Module[2].Input.SkillInput[14].ParameterInput[2] := Module2002.Input.SkillInput.SkillInput14.ParameterInput.ParameterInput2;
Module2002.Output.SkillOutput.SkillOutput14.ParameterOutput.ParameterOutput2 := Module[2].Output.SkillOutput[14].ParameterOutput[2];
Module[2].Input.SkillInput[14].ParameterInput[3] := Module2002.Input.SkillInput.SkillInput14.ParameterInput.ParameterInput3;
Module2002.Output.SkillOutput.SkillOutput14.ParameterOutput.ParameterOutput3 := Module[2].Output.SkillOutput[14].ParameterOutput[3];
Module[2].Input.SkillInput[14].ParameterInput[4] := Module2002.Input.SkillInput.SkillInput14.ParameterInput.ParameterInput4;
Module2002.Output.SkillOutput.SkillOutput14.ParameterOutput.ParameterOutput4 := Module[2].Output.SkillOutput[14].ParameterOutput[4];
Module[2].Input.SkillInput[14].ParameterInput[5] := Module2002.Input.SkillInput.SkillInput14.ParameterInput.ParameterInput5;
Module2002.Output.SkillOutput.SkillOutput14.ParameterOutput.ParameterOutput5 := Module[2].Output.SkillOutput[14].ParameterOutput[5];
Module[2].Input.SkillInput[15].Execute := Module2002.Input.SkillInput.SkillInput15.Execute;
Module2002.Output.SkillOutput.SkillOutput15.Dummy := Module[2].Output.SkillOutput[15].Dummy;
Module2002.Output.SkillOutput.SkillOutput15.ID := Module[2].Output.SkillOutput[15].ID;
Module2002.Output.SkillOutput.SkillOutput15.Name := Module[2].Output.SkillOutput[15].Name;
Module2002.Output.SkillOutput.SkillOutput15.Activated := Module[2].Output.SkillOutput[15].Activated;
Module2002.Output.SkillOutput.SkillOutput15.Ready := Module[2].Output.SkillOutput[15].Ready;
Module2002.Output.SkillOutput.SkillOutput15.Busy := Module[2].Output.SkillOutput[15].Busy;
Module2002.Output.SkillOutput.SkillOutput15.Done := Module[2].Output.SkillOutput[15].Done;
Module2002.Output.SkillOutput.SkillOutput15.Error := Module[2].Output.SkillOutput[15].Error;
Module2002.Output.Statevalue.Statevalue0 := Module[2].Output.Statevalue[0];
Module2002.Output.Statevalue.Statevalue1 := Module[2].Output.Statevalue[1];
Module2002.Output.Statevalue.Statevalue2 := Module[2].Output.Statevalue[2];
Module2002.Output.Statevalue.Statevalue3 := Module[2].Output.Statevalue[3];
Module2002.Output.Statevalue.Statevalue4 := Module[2].Output.Statevalue[4];
Module2002.Output.Statevalue.Statevalue5 := Module[2].Output.Statevalue[5];
Module2002.Output.Statevalue.Statevalue6 := Module[2].Output.Statevalue[6];
Module2002.Output.Statevalue.Statevalue7 := Module[2].Output.Statevalue[7];
Module2002.Output.Statevalue.Statevalue8 := Module[2].Output.Statevalue[8];
Module2002.Output.Statevalue.Statevalue9 := Module[2].Output.Statevalue[9];
Module2002.Output.Statevalue.Statevalue10 := Module[2].Output.Statevalue[10];
Module[2].Input.SkillInput[15].ParameterInput[0] := Module2002.Input.SkillInput.SkillInput15.ParameterInput.ParameterInput0;
Module2002.Output.SkillOutput.SkillOutput15.ParameterOutput.ParameterOutput0 := Module[2].Output.SkillOutput[15].ParameterOutput[0];
Module[2].Input.SkillInput[15].ParameterInput[1] := Module2002.Input.SkillInput.SkillInput15.ParameterInput.ParameterInput1;
Module2002.Output.SkillOutput.SkillOutput15.ParameterOutput.ParameterOutput1 := Module[2].Output.SkillOutput[15].ParameterOutput[1];
Module[2].Input.SkillInput[15].ParameterInput[2] := Module2002.Input.SkillInput.SkillInput15.ParameterInput.ParameterInput2;
Module2002.Output.SkillOutput.SkillOutput15.ParameterOutput.ParameterOutput2 := Module[2].Output.SkillOutput[15].ParameterOutput[2];
Module[2].Input.SkillInput[15].ParameterInput[3] := Module2002.Input.SkillInput.SkillInput15.ParameterInput.ParameterInput3;
Module2002.Output.SkillOutput.SkillOutput15.ParameterOutput.ParameterOutput3 := Module[2].Output.SkillOutput[15].ParameterOutput[3];
Module[2].Input.SkillInput[15].ParameterInput[4] := Module2002.Input.SkillInput.SkillInput15.ParameterInput.ParameterInput4;
Module2002.Output.SkillOutput.SkillOutput15.ParameterOutput.ParameterOutput4 := Module[2].Output.SkillOutput[15].ParameterOutput[4];
Module[2].Input.SkillInput[15].ParameterInput[5] := Module2002.Input.SkillInput.SkillInput15.ParameterInput.ParameterInput5;
Module2002.Output.SkillOutput.SkillOutput15.ParameterOutput.ParameterOutput5 := Module[2].Output.SkillOutput[15].ParameterOutput[5];
Module[3].Input.Mode := Module2003.Input.Mode;
Module[3].Input.ConnectionTestInput := Module2003.Input.ConnectionTestInput;
Module[3].Input.PositionInput := Module2003.Input.PositionInput;
Module[3].Input.Watchbit := Module2003.Input.Watchbit;
Module[3].Input.EmergencyStop := Module2003.Input.EmergencyStop;
Module2003.Output.Dummy := Module[3].Output.Dummy;
Module2003.Output.Name := Module[3].Output.Name;
Module2003.Output.ID := Module[3].Output.ID;
Module2003.Output.IP := Module[3].Output.IP;
Module2003.Output.Idle := Module[3].Output.Idle;
Module2003.Output.Connected := Module[3].Output.Connected;
Module2003.Output.Error := Module[3].Output.Error;
Module2003.Output.ErrorID := Module[3].Output.ErrorID;
Module2003.Output.ErrorDescription := Module[3].Output.ErrorDescription;
Module2003.Output.CurrentTaskDescription := Module[3].Output.CurrentTaskDescription;
Module2003.Output.PositionSensor := Module[3].Output.PositionSensor;
Module2003.Output.ConnectionTestOutput := Module[3].Output.ConnectionTestOutput;
Module[3].Input.SkillInput[0].Execute := Module2003.Input.SkillInput.SkillInput0.Execute;
Module2003.Output.SkillOutput.SkillOutput0.Dummy := Module[3].Output.SkillOutput[0].Dummy;
Module2003.Output.SkillOutput.SkillOutput0.ID := Module[3].Output.SkillOutput[0].ID;
Module2003.Output.SkillOutput.SkillOutput0.Name := Module[3].Output.SkillOutput[0].Name;
Module2003.Output.SkillOutput.SkillOutput0.Activated := Module[3].Output.SkillOutput[0].Activated;
Module2003.Output.SkillOutput.SkillOutput0.Ready := Module[3].Output.SkillOutput[0].Ready;
Module2003.Output.SkillOutput.SkillOutput0.Busy := Module[3].Output.SkillOutput[0].Busy;
Module2003.Output.SkillOutput.SkillOutput0.Done := Module[3].Output.SkillOutput[0].Done;
Module2003.Output.SkillOutput.SkillOutput0.Error := Module[3].Output.SkillOutput[0].Error;
Module2003.Output.Statevalue.Statevalue0 := Module[3].Output.Statevalue[0];
Module2003.Output.Statevalue.Statevalue1 := Module[3].Output.Statevalue[1];
Module2003.Output.Statevalue.Statevalue2 := Module[3].Output.Statevalue[2];
Module2003.Output.Statevalue.Statevalue3 := Module[3].Output.Statevalue[3];
Module2003.Output.Statevalue.Statevalue4 := Module[3].Output.Statevalue[4];
Module2003.Output.Statevalue.Statevalue5 := Module[3].Output.Statevalue[5];
Module2003.Output.Statevalue.Statevalue6 := Module[3].Output.Statevalue[6];
Module2003.Output.Statevalue.Statevalue7 := Module[3].Output.Statevalue[7];
Module2003.Output.Statevalue.Statevalue8 := Module[3].Output.Statevalue[8];
Module2003.Output.Statevalue.Statevalue9 := Module[3].Output.Statevalue[9];
Module2003.Output.Statevalue.Statevalue10 := Module[3].Output.Statevalue[10];
Module[3].Input.SkillInput[0].ParameterInput[0] := Module2003.Input.SkillInput.SkillInput0.ParameterInput.ParameterInput0;
Module2003.Output.SkillOutput.SkillOutput0.ParameterOutput.ParameterOutput0 := Module[3].Output.SkillOutput[0].ParameterOutput[0];
Module[3].Input.SkillInput[0].ParameterInput[1] := Module2003.Input.SkillInput.SkillInput0.ParameterInput.ParameterInput1;
Module2003.Output.SkillOutput.SkillOutput0.ParameterOutput.ParameterOutput1 := Module[3].Output.SkillOutput[0].ParameterOutput[1];
Module[3].Input.SkillInput[0].ParameterInput[2] := Module2003.Input.SkillInput.SkillInput0.ParameterInput.ParameterInput2;
Module2003.Output.SkillOutput.SkillOutput0.ParameterOutput.ParameterOutput2 := Module[3].Output.SkillOutput[0].ParameterOutput[2];
Module[3].Input.SkillInput[0].ParameterInput[3] := Module2003.Input.SkillInput.SkillInput0.ParameterInput.ParameterInput3;
Module2003.Output.SkillOutput.SkillOutput0.ParameterOutput.ParameterOutput3 := Module[3].Output.SkillOutput[0].ParameterOutput[3];
Module[3].Input.SkillInput[0].ParameterInput[4] := Module2003.Input.SkillInput.SkillInput0.ParameterInput.ParameterInput4;
Module2003.Output.SkillOutput.SkillOutput0.ParameterOutput.ParameterOutput4 := Module[3].Output.SkillOutput[0].ParameterOutput[4];
Module[3].Input.SkillInput[0].ParameterInput[5] := Module2003.Input.SkillInput.SkillInput0.ParameterInput.ParameterInput5;
Module2003.Output.SkillOutput.SkillOutput0.ParameterOutput.ParameterOutput5 := Module[3].Output.SkillOutput[0].ParameterOutput[5];
Module[3].Input.SkillInput[1].Execute := Module2003.Input.SkillInput.SkillInput1.Execute;
Module2003.Output.SkillOutput.SkillOutput1.Dummy := Module[3].Output.SkillOutput[1].Dummy;
Module2003.Output.SkillOutput.SkillOutput1.ID := Module[3].Output.SkillOutput[1].ID;
Module2003.Output.SkillOutput.SkillOutput1.Name := Module[3].Output.SkillOutput[1].Name;
Module2003.Output.SkillOutput.SkillOutput1.Activated := Module[3].Output.SkillOutput[1].Activated;
Module2003.Output.SkillOutput.SkillOutput1.Ready := Module[3].Output.SkillOutput[1].Ready;
Module2003.Output.SkillOutput.SkillOutput1.Busy := Module[3].Output.SkillOutput[1].Busy;
Module2003.Output.SkillOutput.SkillOutput1.Done := Module[3].Output.SkillOutput[1].Done;
Module2003.Output.SkillOutput.SkillOutput1.Error := Module[3].Output.SkillOutput[1].Error;
Module2003.Output.Statevalue.Statevalue0 := Module[3].Output.Statevalue[0];
Module2003.Output.Statevalue.Statevalue1 := Module[3].Output.Statevalue[1];
Module2003.Output.Statevalue.Statevalue2 := Module[3].Output.Statevalue[2];
Module2003.Output.Statevalue.Statevalue3 := Module[3].Output.Statevalue[3];
Module2003.Output.Statevalue.Statevalue4 := Module[3].Output.Statevalue[4];
Module2003.Output.Statevalue.Statevalue5 := Module[3].Output.Statevalue[5];
Module2003.Output.Statevalue.Statevalue6 := Module[3].Output.Statevalue[6];
Module2003.Output.Statevalue.Statevalue7 := Module[3].Output.Statevalue[7];
Module2003.Output.Statevalue.Statevalue8 := Module[3].Output.Statevalue[8];
Module2003.Output.Statevalue.Statevalue9 := Module[3].Output.Statevalue[9];
Module2003.Output.Statevalue.Statevalue10 := Module[3].Output.Statevalue[10];
Module[3].Input.SkillInput[1].ParameterInput[0] := Module2003.Input.SkillInput.SkillInput1.ParameterInput.ParameterInput0;
Module2003.Output.SkillOutput.SkillOutput1.ParameterOutput.ParameterOutput0 := Module[3].Output.SkillOutput[1].ParameterOutput[0];
Module[3].Input.SkillInput[1].ParameterInput[1] := Module2003.Input.SkillInput.SkillInput1.ParameterInput.ParameterInput1;
Module2003.Output.SkillOutput.SkillOutput1.ParameterOutput.ParameterOutput1 := Module[3].Output.SkillOutput[1].ParameterOutput[1];
Module[3].Input.SkillInput[1].ParameterInput[2] := Module2003.Input.SkillInput.SkillInput1.ParameterInput.ParameterInput2;
Module2003.Output.SkillOutput.SkillOutput1.ParameterOutput.ParameterOutput2 := Module[3].Output.SkillOutput[1].ParameterOutput[2];
Module[3].Input.SkillInput[1].ParameterInput[3] := Module2003.Input.SkillInput.SkillInput1.ParameterInput.ParameterInput3;
Module2003.Output.SkillOutput.SkillOutput1.ParameterOutput.ParameterOutput3 := Module[3].Output.SkillOutput[1].ParameterOutput[3];
Module[3].Input.SkillInput[1].ParameterInput[4] := Module2003.Input.SkillInput.SkillInput1.ParameterInput.ParameterInput4;
Module2003.Output.SkillOutput.SkillOutput1.ParameterOutput.ParameterOutput4 := Module[3].Output.SkillOutput[1].ParameterOutput[4];
Module[3].Input.SkillInput[1].ParameterInput[5] := Module2003.Input.SkillInput.SkillInput1.ParameterInput.ParameterInput5;
Module2003.Output.SkillOutput.SkillOutput1.ParameterOutput.ParameterOutput5 := Module[3].Output.SkillOutput[1].ParameterOutput[5];
Module[3].Input.SkillInput[2].Execute := Module2003.Input.SkillInput.SkillInput2.Execute;
Module2003.Output.SkillOutput.SkillOutput2.Dummy := Module[3].Output.SkillOutput[2].Dummy;
Module2003.Output.SkillOutput.SkillOutput2.ID := Module[3].Output.SkillOutput[2].ID;
Module2003.Output.SkillOutput.SkillOutput2.Name := Module[3].Output.SkillOutput[2].Name;
Module2003.Output.SkillOutput.SkillOutput2.Activated := Module[3].Output.SkillOutput[2].Activated;
Module2003.Output.SkillOutput.SkillOutput2.Ready := Module[3].Output.SkillOutput[2].Ready;
Module2003.Output.SkillOutput.SkillOutput2.Busy := Module[3].Output.SkillOutput[2].Busy;
Module2003.Output.SkillOutput.SkillOutput2.Done := Module[3].Output.SkillOutput[2].Done;
Module2003.Output.SkillOutput.SkillOutput2.Error := Module[3].Output.SkillOutput[2].Error;
Module2003.Output.Statevalue.Statevalue0 := Module[3].Output.Statevalue[0];
Module2003.Output.Statevalue.Statevalue1 := Module[3].Output.Statevalue[1];
Module2003.Output.Statevalue.Statevalue2 := Module[3].Output.Statevalue[2];
Module2003.Output.Statevalue.Statevalue3 := Module[3].Output.Statevalue[3];
Module2003.Output.Statevalue.Statevalue4 := Module[3].Output.Statevalue[4];
Module2003.Output.Statevalue.Statevalue5 := Module[3].Output.Statevalue[5];
Module2003.Output.Statevalue.Statevalue6 := Module[3].Output.Statevalue[6];
Module2003.Output.Statevalue.Statevalue7 := Module[3].Output.Statevalue[7];
Module2003.Output.Statevalue.Statevalue8 := Module[3].Output.Statevalue[8];
Module2003.Output.Statevalue.Statevalue9 := Module[3].Output.Statevalue[9];
Module2003.Output.Statevalue.Statevalue10 := Module[3].Output.Statevalue[10];
Module[3].Input.SkillInput[2].ParameterInput[0] := Module2003.Input.SkillInput.SkillInput2.ParameterInput.ParameterInput0;
Module2003.Output.SkillOutput.SkillOutput2.ParameterOutput.ParameterOutput0 := Module[3].Output.SkillOutput[2].ParameterOutput[0];
Module[3].Input.SkillInput[2].ParameterInput[1] := Module2003.Input.SkillInput.SkillInput2.ParameterInput.ParameterInput1;
Module2003.Output.SkillOutput.SkillOutput2.ParameterOutput.ParameterOutput1 := Module[3].Output.SkillOutput[2].ParameterOutput[1];
Module[3].Input.SkillInput[2].ParameterInput[2] := Module2003.Input.SkillInput.SkillInput2.ParameterInput.ParameterInput2;
Module2003.Output.SkillOutput.SkillOutput2.ParameterOutput.ParameterOutput2 := Module[3].Output.SkillOutput[2].ParameterOutput[2];
Module[3].Input.SkillInput[2].ParameterInput[3] := Module2003.Input.SkillInput.SkillInput2.ParameterInput.ParameterInput3;
Module2003.Output.SkillOutput.SkillOutput2.ParameterOutput.ParameterOutput3 := Module[3].Output.SkillOutput[2].ParameterOutput[3];
Module[3].Input.SkillInput[2].ParameterInput[4] := Module2003.Input.SkillInput.SkillInput2.ParameterInput.ParameterInput4;
Module2003.Output.SkillOutput.SkillOutput2.ParameterOutput.ParameterOutput4 := Module[3].Output.SkillOutput[2].ParameterOutput[4];
Module[3].Input.SkillInput[2].ParameterInput[5] := Module2003.Input.SkillInput.SkillInput2.ParameterInput.ParameterInput5;
Module2003.Output.SkillOutput.SkillOutput2.ParameterOutput.ParameterOutput5 := Module[3].Output.SkillOutput[2].ParameterOutput[5];
Module[3].Input.SkillInput[3].Execute := Module2003.Input.SkillInput.SkillInput3.Execute;
Module2003.Output.SkillOutput.SkillOutput3.Dummy := Module[3].Output.SkillOutput[3].Dummy;
Module2003.Output.SkillOutput.SkillOutput3.ID := Module[3].Output.SkillOutput[3].ID;
Module2003.Output.SkillOutput.SkillOutput3.Name := Module[3].Output.SkillOutput[3].Name;
Module2003.Output.SkillOutput.SkillOutput3.Activated := Module[3].Output.SkillOutput[3].Activated;
Module2003.Output.SkillOutput.SkillOutput3.Ready := Module[3].Output.SkillOutput[3].Ready;
Module2003.Output.SkillOutput.SkillOutput3.Busy := Module[3].Output.SkillOutput[3].Busy;
Module2003.Output.SkillOutput.SkillOutput3.Done := Module[3].Output.SkillOutput[3].Done;
Module2003.Output.SkillOutput.SkillOutput3.Error := Module[3].Output.SkillOutput[3].Error;
Module2003.Output.Statevalue.Statevalue0 := Module[3].Output.Statevalue[0];
Module2003.Output.Statevalue.Statevalue1 := Module[3].Output.Statevalue[1];
Module2003.Output.Statevalue.Statevalue2 := Module[3].Output.Statevalue[2];
Module2003.Output.Statevalue.Statevalue3 := Module[3].Output.Statevalue[3];
Module2003.Output.Statevalue.Statevalue4 := Module[3].Output.Statevalue[4];
Module2003.Output.Statevalue.Statevalue5 := Module[3].Output.Statevalue[5];
Module2003.Output.Statevalue.Statevalue6 := Module[3].Output.Statevalue[6];
Module2003.Output.Statevalue.Statevalue7 := Module[3].Output.Statevalue[7];
Module2003.Output.Statevalue.Statevalue8 := Module[3].Output.Statevalue[8];
Module2003.Output.Statevalue.Statevalue9 := Module[3].Output.Statevalue[9];
Module2003.Output.Statevalue.Statevalue10 := Module[3].Output.Statevalue[10];
Module[3].Input.SkillInput[3].ParameterInput[0] := Module2003.Input.SkillInput.SkillInput3.ParameterInput.ParameterInput0;
Module2003.Output.SkillOutput.SkillOutput3.ParameterOutput.ParameterOutput0 := Module[3].Output.SkillOutput[3].ParameterOutput[0];
Module[3].Input.SkillInput[3].ParameterInput[1] := Module2003.Input.SkillInput.SkillInput3.ParameterInput.ParameterInput1;
Module2003.Output.SkillOutput.SkillOutput3.ParameterOutput.ParameterOutput1 := Module[3].Output.SkillOutput[3].ParameterOutput[1];
Module[3].Input.SkillInput[3].ParameterInput[2] := Module2003.Input.SkillInput.SkillInput3.ParameterInput.ParameterInput2;
Module2003.Output.SkillOutput.SkillOutput3.ParameterOutput.ParameterOutput2 := Module[3].Output.SkillOutput[3].ParameterOutput[2];
Module[3].Input.SkillInput[3].ParameterInput[3] := Module2003.Input.SkillInput.SkillInput3.ParameterInput.ParameterInput3;
Module2003.Output.SkillOutput.SkillOutput3.ParameterOutput.ParameterOutput3 := Module[3].Output.SkillOutput[3].ParameterOutput[3];
Module[3].Input.SkillInput[3].ParameterInput[4] := Module2003.Input.SkillInput.SkillInput3.ParameterInput.ParameterInput4;
Module2003.Output.SkillOutput.SkillOutput3.ParameterOutput.ParameterOutput4 := Module[3].Output.SkillOutput[3].ParameterOutput[4];
Module[3].Input.SkillInput[3].ParameterInput[5] := Module2003.Input.SkillInput.SkillInput3.ParameterInput.ParameterInput5;
Module2003.Output.SkillOutput.SkillOutput3.ParameterOutput.ParameterOutput5 := Module[3].Output.SkillOutput[3].ParameterOutput[5];
Module[3].Input.SkillInput[4].Execute := Module2003.Input.SkillInput.SkillInput4.Execute;
Module2003.Output.SkillOutput.SkillOutput4.Dummy := Module[3].Output.SkillOutput[4].Dummy;
Module2003.Output.SkillOutput.SkillOutput4.ID := Module[3].Output.SkillOutput[4].ID;
Module2003.Output.SkillOutput.SkillOutput4.Name := Module[3].Output.SkillOutput[4].Name;
Module2003.Output.SkillOutput.SkillOutput4.Activated := Module[3].Output.SkillOutput[4].Activated;
Module2003.Output.SkillOutput.SkillOutput4.Ready := Module[3].Output.SkillOutput[4].Ready;
Module2003.Output.SkillOutput.SkillOutput4.Busy := Module[3].Output.SkillOutput[4].Busy;
Module2003.Output.SkillOutput.SkillOutput4.Done := Module[3].Output.SkillOutput[4].Done;
Module2003.Output.SkillOutput.SkillOutput4.Error := Module[3].Output.SkillOutput[4].Error;
Module2003.Output.Statevalue.Statevalue0 := Module[3].Output.Statevalue[0];
Module2003.Output.Statevalue.Statevalue1 := Module[3].Output.Statevalue[1];
Module2003.Output.Statevalue.Statevalue2 := Module[3].Output.Statevalue[2];
Module2003.Output.Statevalue.Statevalue3 := Module[3].Output.Statevalue[3];
Module2003.Output.Statevalue.Statevalue4 := Module[3].Output.Statevalue[4];
Module2003.Output.Statevalue.Statevalue5 := Module[3].Output.Statevalue[5];
Module2003.Output.Statevalue.Statevalue6 := Module[3].Output.Statevalue[6];
Module2003.Output.Statevalue.Statevalue7 := Module[3].Output.Statevalue[7];
Module2003.Output.Statevalue.Statevalue8 := Module[3].Output.Statevalue[8];
Module2003.Output.Statevalue.Statevalue9 := Module[3].Output.Statevalue[9];
Module2003.Output.Statevalue.Statevalue10 := Module[3].Output.Statevalue[10];
Module[3].Input.SkillInput[4].ParameterInput[0] := Module2003.Input.SkillInput.SkillInput4.ParameterInput.ParameterInput0;
Module2003.Output.SkillOutput.SkillOutput4.ParameterOutput.ParameterOutput0 := Module[3].Output.SkillOutput[4].ParameterOutput[0];
Module[3].Input.SkillInput[4].ParameterInput[1] := Module2003.Input.SkillInput.SkillInput4.ParameterInput.ParameterInput1;
Module2003.Output.SkillOutput.SkillOutput4.ParameterOutput.ParameterOutput1 := Module[3].Output.SkillOutput[4].ParameterOutput[1];
Module[3].Input.SkillInput[4].ParameterInput[2] := Module2003.Input.SkillInput.SkillInput4.ParameterInput.ParameterInput2;
Module2003.Output.SkillOutput.SkillOutput4.ParameterOutput.ParameterOutput2 := Module[3].Output.SkillOutput[4].ParameterOutput[2];
Module[3].Input.SkillInput[4].ParameterInput[3] := Module2003.Input.SkillInput.SkillInput4.ParameterInput.ParameterInput3;
Module2003.Output.SkillOutput.SkillOutput4.ParameterOutput.ParameterOutput3 := Module[3].Output.SkillOutput[4].ParameterOutput[3];
Module[3].Input.SkillInput[4].ParameterInput[4] := Module2003.Input.SkillInput.SkillInput4.ParameterInput.ParameterInput4;
Module2003.Output.SkillOutput.SkillOutput4.ParameterOutput.ParameterOutput4 := Module[3].Output.SkillOutput[4].ParameterOutput[4];
Module[3].Input.SkillInput[4].ParameterInput[5] := Module2003.Input.SkillInput.SkillInput4.ParameterInput.ParameterInput5;
Module2003.Output.SkillOutput.SkillOutput4.ParameterOutput.ParameterOutput5 := Module[3].Output.SkillOutput[4].ParameterOutput[5];
Module[3].Input.SkillInput[5].Execute := Module2003.Input.SkillInput.SkillInput5.Execute;
Module2003.Output.SkillOutput.SkillOutput5.Dummy := Module[3].Output.SkillOutput[5].Dummy;
Module2003.Output.SkillOutput.SkillOutput5.ID := Module[3].Output.SkillOutput[5].ID;
Module2003.Output.SkillOutput.SkillOutput5.Name := Module[3].Output.SkillOutput[5].Name;
Module2003.Output.SkillOutput.SkillOutput5.Activated := Module[3].Output.SkillOutput[5].Activated;
Module2003.Output.SkillOutput.SkillOutput5.Ready := Module[3].Output.SkillOutput[5].Ready;
Module2003.Output.SkillOutput.SkillOutput5.Busy := Module[3].Output.SkillOutput[5].Busy;
Module2003.Output.SkillOutput.SkillOutput5.Done := Module[3].Output.SkillOutput[5].Done;
Module2003.Output.SkillOutput.SkillOutput5.Error := Module[3].Output.SkillOutput[5].Error;
Module2003.Output.Statevalue.Statevalue0 := Module[3].Output.Statevalue[0];
Module2003.Output.Statevalue.Statevalue1 := Module[3].Output.Statevalue[1];
Module2003.Output.Statevalue.Statevalue2 := Module[3].Output.Statevalue[2];
Module2003.Output.Statevalue.Statevalue3 := Module[3].Output.Statevalue[3];
Module2003.Output.Statevalue.Statevalue4 := Module[3].Output.Statevalue[4];
Module2003.Output.Statevalue.Statevalue5 := Module[3].Output.Statevalue[5];
Module2003.Output.Statevalue.Statevalue6 := Module[3].Output.Statevalue[6];
Module2003.Output.Statevalue.Statevalue7 := Module[3].Output.Statevalue[7];
Module2003.Output.Statevalue.Statevalue8 := Module[3].Output.Statevalue[8];
Module2003.Output.Statevalue.Statevalue9 := Module[3].Output.Statevalue[9];
Module2003.Output.Statevalue.Statevalue10 := Module[3].Output.Statevalue[10];
Module[3].Input.SkillInput[5].ParameterInput[0] := Module2003.Input.SkillInput.SkillInput5.ParameterInput.ParameterInput0;
Module2003.Output.SkillOutput.SkillOutput5.ParameterOutput.ParameterOutput0 := Module[3].Output.SkillOutput[5].ParameterOutput[0];
Module[3].Input.SkillInput[5].ParameterInput[1] := Module2003.Input.SkillInput.SkillInput5.ParameterInput.ParameterInput1;
Module2003.Output.SkillOutput.SkillOutput5.ParameterOutput.ParameterOutput1 := Module[3].Output.SkillOutput[5].ParameterOutput[1];
Module[3].Input.SkillInput[5].ParameterInput[2] := Module2003.Input.SkillInput.SkillInput5.ParameterInput.ParameterInput2;
Module2003.Output.SkillOutput.SkillOutput5.ParameterOutput.ParameterOutput2 := Module[3].Output.SkillOutput[5].ParameterOutput[2];
Module[3].Input.SkillInput[5].ParameterInput[3] := Module2003.Input.SkillInput.SkillInput5.ParameterInput.ParameterInput3;
Module2003.Output.SkillOutput.SkillOutput5.ParameterOutput.ParameterOutput3 := Module[3].Output.SkillOutput[5].ParameterOutput[3];
Module[3].Input.SkillInput[5].ParameterInput[4] := Module2003.Input.SkillInput.SkillInput5.ParameterInput.ParameterInput4;
Module2003.Output.SkillOutput.SkillOutput5.ParameterOutput.ParameterOutput4 := Module[3].Output.SkillOutput[5].ParameterOutput[4];
Module[3].Input.SkillInput[5].ParameterInput[5] := Module2003.Input.SkillInput.SkillInput5.ParameterInput.ParameterInput5;
Module2003.Output.SkillOutput.SkillOutput5.ParameterOutput.ParameterOutput5 := Module[3].Output.SkillOutput[5].ParameterOutput[5];
Module[3].Input.SkillInput[6].Execute := Module2003.Input.SkillInput.SkillInput6.Execute;
Module2003.Output.SkillOutput.SkillOutput6.Dummy := Module[3].Output.SkillOutput[6].Dummy;
Module2003.Output.SkillOutput.SkillOutput6.ID := Module[3].Output.SkillOutput[6].ID;
Module2003.Output.SkillOutput.SkillOutput6.Name := Module[3].Output.SkillOutput[6].Name;
Module2003.Output.SkillOutput.SkillOutput6.Activated := Module[3].Output.SkillOutput[6].Activated;
Module2003.Output.SkillOutput.SkillOutput6.Ready := Module[3].Output.SkillOutput[6].Ready;
Module2003.Output.SkillOutput.SkillOutput6.Busy := Module[3].Output.SkillOutput[6].Busy;
Module2003.Output.SkillOutput.SkillOutput6.Done := Module[3].Output.SkillOutput[6].Done;
Module2003.Output.SkillOutput.SkillOutput6.Error := Module[3].Output.SkillOutput[6].Error;
Module2003.Output.Statevalue.Statevalue0 := Module[3].Output.Statevalue[0];
Module2003.Output.Statevalue.Statevalue1 := Module[3].Output.Statevalue[1];
Module2003.Output.Statevalue.Statevalue2 := Module[3].Output.Statevalue[2];
Module2003.Output.Statevalue.Statevalue3 := Module[3].Output.Statevalue[3];
Module2003.Output.Statevalue.Statevalue4 := Module[3].Output.Statevalue[4];
Module2003.Output.Statevalue.Statevalue5 := Module[3].Output.Statevalue[5];
Module2003.Output.Statevalue.Statevalue6 := Module[3].Output.Statevalue[6];
Module2003.Output.Statevalue.Statevalue7 := Module[3].Output.Statevalue[7];
Module2003.Output.Statevalue.Statevalue8 := Module[3].Output.Statevalue[8];
Module2003.Output.Statevalue.Statevalue9 := Module[3].Output.Statevalue[9];
Module2003.Output.Statevalue.Statevalue10 := Module[3].Output.Statevalue[10];
Module[3].Input.SkillInput[6].ParameterInput[0] := Module2003.Input.SkillInput.SkillInput6.ParameterInput.ParameterInput0;
Module2003.Output.SkillOutput.SkillOutput6.ParameterOutput.ParameterOutput0 := Module[3].Output.SkillOutput[6].ParameterOutput[0];
Module[3].Input.SkillInput[6].ParameterInput[1] := Module2003.Input.SkillInput.SkillInput6.ParameterInput.ParameterInput1;
Module2003.Output.SkillOutput.SkillOutput6.ParameterOutput.ParameterOutput1 := Module[3].Output.SkillOutput[6].ParameterOutput[1];
Module[3].Input.SkillInput[6].ParameterInput[2] := Module2003.Input.SkillInput.SkillInput6.ParameterInput.ParameterInput2;
Module2003.Output.SkillOutput.SkillOutput6.ParameterOutput.ParameterOutput2 := Module[3].Output.SkillOutput[6].ParameterOutput[2];
Module[3].Input.SkillInput[6].ParameterInput[3] := Module2003.Input.SkillInput.SkillInput6.ParameterInput.ParameterInput3;
Module2003.Output.SkillOutput.SkillOutput6.ParameterOutput.ParameterOutput3 := Module[3].Output.SkillOutput[6].ParameterOutput[3];
Module[3].Input.SkillInput[6].ParameterInput[4] := Module2003.Input.SkillInput.SkillInput6.ParameterInput.ParameterInput4;
Module2003.Output.SkillOutput.SkillOutput6.ParameterOutput.ParameterOutput4 := Module[3].Output.SkillOutput[6].ParameterOutput[4];
Module[3].Input.SkillInput[6].ParameterInput[5] := Module2003.Input.SkillInput.SkillInput6.ParameterInput.ParameterInput5;
Module2003.Output.SkillOutput.SkillOutput6.ParameterOutput.ParameterOutput5 := Module[3].Output.SkillOutput[6].ParameterOutput[5];
Module[3].Input.SkillInput[7].Execute := Module2003.Input.SkillInput.SkillInput7.Execute;
Module2003.Output.SkillOutput.SkillOutput7.Dummy := Module[3].Output.SkillOutput[7].Dummy;
Module2003.Output.SkillOutput.SkillOutput7.ID := Module[3].Output.SkillOutput[7].ID;
Module2003.Output.SkillOutput.SkillOutput7.Name := Module[3].Output.SkillOutput[7].Name;
Module2003.Output.SkillOutput.SkillOutput7.Activated := Module[3].Output.SkillOutput[7].Activated;
Module2003.Output.SkillOutput.SkillOutput7.Ready := Module[3].Output.SkillOutput[7].Ready;
Module2003.Output.SkillOutput.SkillOutput7.Busy := Module[3].Output.SkillOutput[7].Busy;
Module2003.Output.SkillOutput.SkillOutput7.Done := Module[3].Output.SkillOutput[7].Done;
Module2003.Output.SkillOutput.SkillOutput7.Error := Module[3].Output.SkillOutput[7].Error;
Module2003.Output.Statevalue.Statevalue0 := Module[3].Output.Statevalue[0];
Module2003.Output.Statevalue.Statevalue1 := Module[3].Output.Statevalue[1];
Module2003.Output.Statevalue.Statevalue2 := Module[3].Output.Statevalue[2];
Module2003.Output.Statevalue.Statevalue3 := Module[3].Output.Statevalue[3];
Module2003.Output.Statevalue.Statevalue4 := Module[3].Output.Statevalue[4];
Module2003.Output.Statevalue.Statevalue5 := Module[3].Output.Statevalue[5];
Module2003.Output.Statevalue.Statevalue6 := Module[3].Output.Statevalue[6];
Module2003.Output.Statevalue.Statevalue7 := Module[3].Output.Statevalue[7];
Module2003.Output.Statevalue.Statevalue8 := Module[3].Output.Statevalue[8];
Module2003.Output.Statevalue.Statevalue9 := Module[3].Output.Statevalue[9];
Module2003.Output.Statevalue.Statevalue10 := Module[3].Output.Statevalue[10];
Module[3].Input.SkillInput[7].ParameterInput[0] := Module2003.Input.SkillInput.SkillInput7.ParameterInput.ParameterInput0;
Module2003.Output.SkillOutput.SkillOutput7.ParameterOutput.ParameterOutput0 := Module[3].Output.SkillOutput[7].ParameterOutput[0];
Module[3].Input.SkillInput[7].ParameterInput[1] := Module2003.Input.SkillInput.SkillInput7.ParameterInput.ParameterInput1;
Module2003.Output.SkillOutput.SkillOutput7.ParameterOutput.ParameterOutput1 := Module[3].Output.SkillOutput[7].ParameterOutput[1];
Module[3].Input.SkillInput[7].ParameterInput[2] := Module2003.Input.SkillInput.SkillInput7.ParameterInput.ParameterInput2;
Module2003.Output.SkillOutput.SkillOutput7.ParameterOutput.ParameterOutput2 := Module[3].Output.SkillOutput[7].ParameterOutput[2];
Module[3].Input.SkillInput[7].ParameterInput[3] := Module2003.Input.SkillInput.SkillInput7.ParameterInput.ParameterInput3;
Module2003.Output.SkillOutput.SkillOutput7.ParameterOutput.ParameterOutput3 := Module[3].Output.SkillOutput[7].ParameterOutput[3];
Module[3].Input.SkillInput[7].ParameterInput[4] := Module2003.Input.SkillInput.SkillInput7.ParameterInput.ParameterInput4;
Module2003.Output.SkillOutput.SkillOutput7.ParameterOutput.ParameterOutput4 := Module[3].Output.SkillOutput[7].ParameterOutput[4];
Module[3].Input.SkillInput[7].ParameterInput[5] := Module2003.Input.SkillInput.SkillInput7.ParameterInput.ParameterInput5;
Module2003.Output.SkillOutput.SkillOutput7.ParameterOutput.ParameterOutput5 := Module[3].Output.SkillOutput[7].ParameterOutput[5];
Module[3].Input.SkillInput[8].Execute := Module2003.Input.SkillInput.SkillInput8.Execute;
Module2003.Output.SkillOutput.SkillOutput8.Dummy := Module[3].Output.SkillOutput[8].Dummy;
Module2003.Output.SkillOutput.SkillOutput8.ID := Module[3].Output.SkillOutput[8].ID;
Module2003.Output.SkillOutput.SkillOutput8.Name := Module[3].Output.SkillOutput[8].Name;
Module2003.Output.SkillOutput.SkillOutput8.Activated := Module[3].Output.SkillOutput[8].Activated;
Module2003.Output.SkillOutput.SkillOutput8.Ready := Module[3].Output.SkillOutput[8].Ready;
Module2003.Output.SkillOutput.SkillOutput8.Busy := Module[3].Output.SkillOutput[8].Busy;
Module2003.Output.SkillOutput.SkillOutput8.Done := Module[3].Output.SkillOutput[8].Done;
Module2003.Output.SkillOutput.SkillOutput8.Error := Module[3].Output.SkillOutput[8].Error;
Module2003.Output.Statevalue.Statevalue0 := Module[3].Output.Statevalue[0];
Module2003.Output.Statevalue.Statevalue1 := Module[3].Output.Statevalue[1];
Module2003.Output.Statevalue.Statevalue2 := Module[3].Output.Statevalue[2];
Module2003.Output.Statevalue.Statevalue3 := Module[3].Output.Statevalue[3];
Module2003.Output.Statevalue.Statevalue4 := Module[3].Output.Statevalue[4];
Module2003.Output.Statevalue.Statevalue5 := Module[3].Output.Statevalue[5];
Module2003.Output.Statevalue.Statevalue6 := Module[3].Output.Statevalue[6];
Module2003.Output.Statevalue.Statevalue7 := Module[3].Output.Statevalue[7];
Module2003.Output.Statevalue.Statevalue8 := Module[3].Output.Statevalue[8];
Module2003.Output.Statevalue.Statevalue9 := Module[3].Output.Statevalue[9];
Module2003.Output.Statevalue.Statevalue10 := Module[3].Output.Statevalue[10];
Module[3].Input.SkillInput[8].ParameterInput[0] := Module2003.Input.SkillInput.SkillInput8.ParameterInput.ParameterInput0;
Module2003.Output.SkillOutput.SkillOutput8.ParameterOutput.ParameterOutput0 := Module[3].Output.SkillOutput[8].ParameterOutput[0];
Module[3].Input.SkillInput[8].ParameterInput[1] := Module2003.Input.SkillInput.SkillInput8.ParameterInput.ParameterInput1;
Module2003.Output.SkillOutput.SkillOutput8.ParameterOutput.ParameterOutput1 := Module[3].Output.SkillOutput[8].ParameterOutput[1];
Module[3].Input.SkillInput[8].ParameterInput[2] := Module2003.Input.SkillInput.SkillInput8.ParameterInput.ParameterInput2;
Module2003.Output.SkillOutput.SkillOutput8.ParameterOutput.ParameterOutput2 := Module[3].Output.SkillOutput[8].ParameterOutput[2];
Module[3].Input.SkillInput[8].ParameterInput[3] := Module2003.Input.SkillInput.SkillInput8.ParameterInput.ParameterInput3;
Module2003.Output.SkillOutput.SkillOutput8.ParameterOutput.ParameterOutput3 := Module[3].Output.SkillOutput[8].ParameterOutput[3];
Module[3].Input.SkillInput[8].ParameterInput[4] := Module2003.Input.SkillInput.SkillInput8.ParameterInput.ParameterInput4;
Module2003.Output.SkillOutput.SkillOutput8.ParameterOutput.ParameterOutput4 := Module[3].Output.SkillOutput[8].ParameterOutput[4];
Module[3].Input.SkillInput[8].ParameterInput[5] := Module2003.Input.SkillInput.SkillInput8.ParameterInput.ParameterInput5;
Module2003.Output.SkillOutput.SkillOutput8.ParameterOutput.ParameterOutput5 := Module[3].Output.SkillOutput[8].ParameterOutput[5];
Module[3].Input.SkillInput[9].Execute := Module2003.Input.SkillInput.SkillInput9.Execute;
Module2003.Output.SkillOutput.SkillOutput9.Dummy := Module[3].Output.SkillOutput[9].Dummy;
Module2003.Output.SkillOutput.SkillOutput9.ID := Module[3].Output.SkillOutput[9].ID;
Module2003.Output.SkillOutput.SkillOutput9.Name := Module[3].Output.SkillOutput[9].Name;
Module2003.Output.SkillOutput.SkillOutput9.Activated := Module[3].Output.SkillOutput[9].Activated;
Module2003.Output.SkillOutput.SkillOutput9.Ready := Module[3].Output.SkillOutput[9].Ready;
Module2003.Output.SkillOutput.SkillOutput9.Busy := Module[3].Output.SkillOutput[9].Busy;
Module2003.Output.SkillOutput.SkillOutput9.Done := Module[3].Output.SkillOutput[9].Done;
Module2003.Output.SkillOutput.SkillOutput9.Error := Module[3].Output.SkillOutput[9].Error;
Module2003.Output.Statevalue.Statevalue0 := Module[3].Output.Statevalue[0];
Module2003.Output.Statevalue.Statevalue1 := Module[3].Output.Statevalue[1];
Module2003.Output.Statevalue.Statevalue2 := Module[3].Output.Statevalue[2];
Module2003.Output.Statevalue.Statevalue3 := Module[3].Output.Statevalue[3];
Module2003.Output.Statevalue.Statevalue4 := Module[3].Output.Statevalue[4];
Module2003.Output.Statevalue.Statevalue5 := Module[3].Output.Statevalue[5];
Module2003.Output.Statevalue.Statevalue6 := Module[3].Output.Statevalue[6];
Module2003.Output.Statevalue.Statevalue7 := Module[3].Output.Statevalue[7];
Module2003.Output.Statevalue.Statevalue8 := Module[3].Output.Statevalue[8];
Module2003.Output.Statevalue.Statevalue9 := Module[3].Output.Statevalue[9];
Module2003.Output.Statevalue.Statevalue10 := Module[3].Output.Statevalue[10];
Module[3].Input.SkillInput[9].ParameterInput[0] := Module2003.Input.SkillInput.SkillInput9.ParameterInput.ParameterInput0;
Module2003.Output.SkillOutput.SkillOutput9.ParameterOutput.ParameterOutput0 := Module[3].Output.SkillOutput[9].ParameterOutput[0];
Module[3].Input.SkillInput[9].ParameterInput[1] := Module2003.Input.SkillInput.SkillInput9.ParameterInput.ParameterInput1;
Module2003.Output.SkillOutput.SkillOutput9.ParameterOutput.ParameterOutput1 := Module[3].Output.SkillOutput[9].ParameterOutput[1];
Module[3].Input.SkillInput[9].ParameterInput[2] := Module2003.Input.SkillInput.SkillInput9.ParameterInput.ParameterInput2;
Module2003.Output.SkillOutput.SkillOutput9.ParameterOutput.ParameterOutput2 := Module[3].Output.SkillOutput[9].ParameterOutput[2];
Module[3].Input.SkillInput[9].ParameterInput[3] := Module2003.Input.SkillInput.SkillInput9.ParameterInput.ParameterInput3;
Module2003.Output.SkillOutput.SkillOutput9.ParameterOutput.ParameterOutput3 := Module[3].Output.SkillOutput[9].ParameterOutput[3];
Module[3].Input.SkillInput[9].ParameterInput[4] := Module2003.Input.SkillInput.SkillInput9.ParameterInput.ParameterInput4;
Module2003.Output.SkillOutput.SkillOutput9.ParameterOutput.ParameterOutput4 := Module[3].Output.SkillOutput[9].ParameterOutput[4];
Module[3].Input.SkillInput[9].ParameterInput[5] := Module2003.Input.SkillInput.SkillInput9.ParameterInput.ParameterInput5;
Module2003.Output.SkillOutput.SkillOutput9.ParameterOutput.ParameterOutput5 := Module[3].Output.SkillOutput[9].ParameterOutput[5];
Module[3].Input.SkillInput[10].Execute := Module2003.Input.SkillInput.SkillInput10.Execute;
Module2003.Output.SkillOutput.SkillOutput10.Dummy := Module[3].Output.SkillOutput[10].Dummy;
Module2003.Output.SkillOutput.SkillOutput10.ID := Module[3].Output.SkillOutput[10].ID;
Module2003.Output.SkillOutput.SkillOutput10.Name := Module[3].Output.SkillOutput[10].Name;
Module2003.Output.SkillOutput.SkillOutput10.Activated := Module[3].Output.SkillOutput[10].Activated;
Module2003.Output.SkillOutput.SkillOutput10.Ready := Module[3].Output.SkillOutput[10].Ready;
Module2003.Output.SkillOutput.SkillOutput10.Busy := Module[3].Output.SkillOutput[10].Busy;
Module2003.Output.SkillOutput.SkillOutput10.Done := Module[3].Output.SkillOutput[10].Done;
Module2003.Output.SkillOutput.SkillOutput10.Error := Module[3].Output.SkillOutput[10].Error;
Module2003.Output.Statevalue.Statevalue0 := Module[3].Output.Statevalue[0];
Module2003.Output.Statevalue.Statevalue1 := Module[3].Output.Statevalue[1];
Module2003.Output.Statevalue.Statevalue2 := Module[3].Output.Statevalue[2];
Module2003.Output.Statevalue.Statevalue3 := Module[3].Output.Statevalue[3];
Module2003.Output.Statevalue.Statevalue4 := Module[3].Output.Statevalue[4];
Module2003.Output.Statevalue.Statevalue5 := Module[3].Output.Statevalue[5];
Module2003.Output.Statevalue.Statevalue6 := Module[3].Output.Statevalue[6];
Module2003.Output.Statevalue.Statevalue7 := Module[3].Output.Statevalue[7];
Module2003.Output.Statevalue.Statevalue8 := Module[3].Output.Statevalue[8];
Module2003.Output.Statevalue.Statevalue9 := Module[3].Output.Statevalue[9];
Module2003.Output.Statevalue.Statevalue10 := Module[3].Output.Statevalue[10];
Module[3].Input.SkillInput[10].ParameterInput[0] := Module2003.Input.SkillInput.SkillInput10.ParameterInput.ParameterInput0;
Module2003.Output.SkillOutput.SkillOutput10.ParameterOutput.ParameterOutput0 := Module[3].Output.SkillOutput[10].ParameterOutput[0];
Module[3].Input.SkillInput[10].ParameterInput[1] := Module2003.Input.SkillInput.SkillInput10.ParameterInput.ParameterInput1;
Module2003.Output.SkillOutput.SkillOutput10.ParameterOutput.ParameterOutput1 := Module[3].Output.SkillOutput[10].ParameterOutput[1];
Module[3].Input.SkillInput[10].ParameterInput[2] := Module2003.Input.SkillInput.SkillInput10.ParameterInput.ParameterInput2;
Module2003.Output.SkillOutput.SkillOutput10.ParameterOutput.ParameterOutput2 := Module[3].Output.SkillOutput[10].ParameterOutput[2];
Module[3].Input.SkillInput[10].ParameterInput[3] := Module2003.Input.SkillInput.SkillInput10.ParameterInput.ParameterInput3;
Module2003.Output.SkillOutput.SkillOutput10.ParameterOutput.ParameterOutput3 := Module[3].Output.SkillOutput[10].ParameterOutput[3];
Module[3].Input.SkillInput[10].ParameterInput[4] := Module2003.Input.SkillInput.SkillInput10.ParameterInput.ParameterInput4;
Module2003.Output.SkillOutput.SkillOutput10.ParameterOutput.ParameterOutput4 := Module[3].Output.SkillOutput[10].ParameterOutput[4];
Module[3].Input.SkillInput[10].ParameterInput[5] := Module2003.Input.SkillInput.SkillInput10.ParameterInput.ParameterInput5;
Module2003.Output.SkillOutput.SkillOutput10.ParameterOutput.ParameterOutput5 := Module[3].Output.SkillOutput[10].ParameterOutput[5];
Module[3].Input.SkillInput[11].Execute := Module2003.Input.SkillInput.SkillInput11.Execute;
Module2003.Output.SkillOutput.SkillOutput11.Dummy := Module[3].Output.SkillOutput[11].Dummy;
Module2003.Output.SkillOutput.SkillOutput11.ID := Module[3].Output.SkillOutput[11].ID;
Module2003.Output.SkillOutput.SkillOutput11.Name := Module[3].Output.SkillOutput[11].Name;
Module2003.Output.SkillOutput.SkillOutput11.Activated := Module[3].Output.SkillOutput[11].Activated;
Module2003.Output.SkillOutput.SkillOutput11.Ready := Module[3].Output.SkillOutput[11].Ready;
Module2003.Output.SkillOutput.SkillOutput11.Busy := Module[3].Output.SkillOutput[11].Busy;
Module2003.Output.SkillOutput.SkillOutput11.Done := Module[3].Output.SkillOutput[11].Done;
Module2003.Output.SkillOutput.SkillOutput11.Error := Module[3].Output.SkillOutput[11].Error;
Module2003.Output.Statevalue.Statevalue0 := Module[3].Output.Statevalue[0];
Module2003.Output.Statevalue.Statevalue1 := Module[3].Output.Statevalue[1];
Module2003.Output.Statevalue.Statevalue2 := Module[3].Output.Statevalue[2];
Module2003.Output.Statevalue.Statevalue3 := Module[3].Output.Statevalue[3];
Module2003.Output.Statevalue.Statevalue4 := Module[3].Output.Statevalue[4];
Module2003.Output.Statevalue.Statevalue5 := Module[3].Output.Statevalue[5];
Module2003.Output.Statevalue.Statevalue6 := Module[3].Output.Statevalue[6];
Module2003.Output.Statevalue.Statevalue7 := Module[3].Output.Statevalue[7];
Module2003.Output.Statevalue.Statevalue8 := Module[3].Output.Statevalue[8];
Module2003.Output.Statevalue.Statevalue9 := Module[3].Output.Statevalue[9];
Module2003.Output.Statevalue.Statevalue10 := Module[3].Output.Statevalue[10];
Module[3].Input.SkillInput[11].ParameterInput[0] := Module2003.Input.SkillInput.SkillInput11.ParameterInput.ParameterInput0;
Module2003.Output.SkillOutput.SkillOutput11.ParameterOutput.ParameterOutput0 := Module[3].Output.SkillOutput[11].ParameterOutput[0];
Module[3].Input.SkillInput[11].ParameterInput[1] := Module2003.Input.SkillInput.SkillInput11.ParameterInput.ParameterInput1;
Module2003.Output.SkillOutput.SkillOutput11.ParameterOutput.ParameterOutput1 := Module[3].Output.SkillOutput[11].ParameterOutput[1];
Module[3].Input.SkillInput[11].ParameterInput[2] := Module2003.Input.SkillInput.SkillInput11.ParameterInput.ParameterInput2;
Module2003.Output.SkillOutput.SkillOutput11.ParameterOutput.ParameterOutput2 := Module[3].Output.SkillOutput[11].ParameterOutput[2];
Module[3].Input.SkillInput[11].ParameterInput[3] := Module2003.Input.SkillInput.SkillInput11.ParameterInput.ParameterInput3;
Module2003.Output.SkillOutput.SkillOutput11.ParameterOutput.ParameterOutput3 := Module[3].Output.SkillOutput[11].ParameterOutput[3];
Module[3].Input.SkillInput[11].ParameterInput[4] := Module2003.Input.SkillInput.SkillInput11.ParameterInput.ParameterInput4;
Module2003.Output.SkillOutput.SkillOutput11.ParameterOutput.ParameterOutput4 := Module[3].Output.SkillOutput[11].ParameterOutput[4];
Module[3].Input.SkillInput[11].ParameterInput[5] := Module2003.Input.SkillInput.SkillInput11.ParameterInput.ParameterInput5;
Module2003.Output.SkillOutput.SkillOutput11.ParameterOutput.ParameterOutput5 := Module[3].Output.SkillOutput[11].ParameterOutput[5];
Module[3].Input.SkillInput[12].Execute := Module2003.Input.SkillInput.SkillInput12.Execute;
Module2003.Output.SkillOutput.SkillOutput12.Dummy := Module[3].Output.SkillOutput[12].Dummy;
Module2003.Output.SkillOutput.SkillOutput12.ID := Module[3].Output.SkillOutput[12].ID;
Module2003.Output.SkillOutput.SkillOutput12.Name := Module[3].Output.SkillOutput[12].Name;
Module2003.Output.SkillOutput.SkillOutput12.Activated := Module[3].Output.SkillOutput[12].Activated;
Module2003.Output.SkillOutput.SkillOutput12.Ready := Module[3].Output.SkillOutput[12].Ready;
Module2003.Output.SkillOutput.SkillOutput12.Busy := Module[3].Output.SkillOutput[12].Busy;
Module2003.Output.SkillOutput.SkillOutput12.Done := Module[3].Output.SkillOutput[12].Done;
Module2003.Output.SkillOutput.SkillOutput12.Error := Module[3].Output.SkillOutput[12].Error;
Module2003.Output.Statevalue.Statevalue0 := Module[3].Output.Statevalue[0];
Module2003.Output.Statevalue.Statevalue1 := Module[3].Output.Statevalue[1];
Module2003.Output.Statevalue.Statevalue2 := Module[3].Output.Statevalue[2];
Module2003.Output.Statevalue.Statevalue3 := Module[3].Output.Statevalue[3];
Module2003.Output.Statevalue.Statevalue4 := Module[3].Output.Statevalue[4];
Module2003.Output.Statevalue.Statevalue5 := Module[3].Output.Statevalue[5];
Module2003.Output.Statevalue.Statevalue6 := Module[3].Output.Statevalue[6];
Module2003.Output.Statevalue.Statevalue7 := Module[3].Output.Statevalue[7];
Module2003.Output.Statevalue.Statevalue8 := Module[3].Output.Statevalue[8];
Module2003.Output.Statevalue.Statevalue9 := Module[3].Output.Statevalue[9];
Module2003.Output.Statevalue.Statevalue10 := Module[3].Output.Statevalue[10];
Module[3].Input.SkillInput[12].ParameterInput[0] := Module2003.Input.SkillInput.SkillInput12.ParameterInput.ParameterInput0;
Module2003.Output.SkillOutput.SkillOutput12.ParameterOutput.ParameterOutput0 := Module[3].Output.SkillOutput[12].ParameterOutput[0];
Module[3].Input.SkillInput[12].ParameterInput[1] := Module2003.Input.SkillInput.SkillInput12.ParameterInput.ParameterInput1;
Module2003.Output.SkillOutput.SkillOutput12.ParameterOutput.ParameterOutput1 := Module[3].Output.SkillOutput[12].ParameterOutput[1];
Module[3].Input.SkillInput[12].ParameterInput[2] := Module2003.Input.SkillInput.SkillInput12.ParameterInput.ParameterInput2;
Module2003.Output.SkillOutput.SkillOutput12.ParameterOutput.ParameterOutput2 := Module[3].Output.SkillOutput[12].ParameterOutput[2];
Module[3].Input.SkillInput[12].ParameterInput[3] := Module2003.Input.SkillInput.SkillInput12.ParameterInput.ParameterInput3;
Module2003.Output.SkillOutput.SkillOutput12.ParameterOutput.ParameterOutput3 := Module[3].Output.SkillOutput[12].ParameterOutput[3];
Module[3].Input.SkillInput[12].ParameterInput[4] := Module2003.Input.SkillInput.SkillInput12.ParameterInput.ParameterInput4;
Module2003.Output.SkillOutput.SkillOutput12.ParameterOutput.ParameterOutput4 := Module[3].Output.SkillOutput[12].ParameterOutput[4];
Module[3].Input.SkillInput[12].ParameterInput[5] := Module2003.Input.SkillInput.SkillInput12.ParameterInput.ParameterInput5;
Module2003.Output.SkillOutput.SkillOutput12.ParameterOutput.ParameterOutput5 := Module[3].Output.SkillOutput[12].ParameterOutput[5];
Module[3].Input.SkillInput[13].Execute := Module2003.Input.SkillInput.SkillInput13.Execute;
Module2003.Output.SkillOutput.SkillOutput13.Dummy := Module[3].Output.SkillOutput[13].Dummy;
Module2003.Output.SkillOutput.SkillOutput13.ID := Module[3].Output.SkillOutput[13].ID;
Module2003.Output.SkillOutput.SkillOutput13.Name := Module[3].Output.SkillOutput[13].Name;
Module2003.Output.SkillOutput.SkillOutput13.Activated := Module[3].Output.SkillOutput[13].Activated;
Module2003.Output.SkillOutput.SkillOutput13.Ready := Module[3].Output.SkillOutput[13].Ready;
Module2003.Output.SkillOutput.SkillOutput13.Busy := Module[3].Output.SkillOutput[13].Busy;
Module2003.Output.SkillOutput.SkillOutput13.Done := Module[3].Output.SkillOutput[13].Done;
Module2003.Output.SkillOutput.SkillOutput13.Error := Module[3].Output.SkillOutput[13].Error;
Module2003.Output.Statevalue.Statevalue0 := Module[3].Output.Statevalue[0];
Module2003.Output.Statevalue.Statevalue1 := Module[3].Output.Statevalue[1];
Module2003.Output.Statevalue.Statevalue2 := Module[3].Output.Statevalue[2];
Module2003.Output.Statevalue.Statevalue3 := Module[3].Output.Statevalue[3];
Module2003.Output.Statevalue.Statevalue4 := Module[3].Output.Statevalue[4];
Module2003.Output.Statevalue.Statevalue5 := Module[3].Output.Statevalue[5];
Module2003.Output.Statevalue.Statevalue6 := Module[3].Output.Statevalue[6];
Module2003.Output.Statevalue.Statevalue7 := Module[3].Output.Statevalue[7];
Module2003.Output.Statevalue.Statevalue8 := Module[3].Output.Statevalue[8];
Module2003.Output.Statevalue.Statevalue9 := Module[3].Output.Statevalue[9];
Module2003.Output.Statevalue.Statevalue10 := Module[3].Output.Statevalue[10];
Module[3].Input.SkillInput[13].ParameterInput[0] := Module2003.Input.SkillInput.SkillInput13.ParameterInput.ParameterInput0;
Module2003.Output.SkillOutput.SkillOutput13.ParameterOutput.ParameterOutput0 := Module[3].Output.SkillOutput[13].ParameterOutput[0];
Module[3].Input.SkillInput[13].ParameterInput[1] := Module2003.Input.SkillInput.SkillInput13.ParameterInput.ParameterInput1;
Module2003.Output.SkillOutput.SkillOutput13.ParameterOutput.ParameterOutput1 := Module[3].Output.SkillOutput[13].ParameterOutput[1];
Module[3].Input.SkillInput[13].ParameterInput[2] := Module2003.Input.SkillInput.SkillInput13.ParameterInput.ParameterInput2;
Module2003.Output.SkillOutput.SkillOutput13.ParameterOutput.ParameterOutput2 := Module[3].Output.SkillOutput[13].ParameterOutput[2];
Module[3].Input.SkillInput[13].ParameterInput[3] := Module2003.Input.SkillInput.SkillInput13.ParameterInput.ParameterInput3;
Module2003.Output.SkillOutput.SkillOutput13.ParameterOutput.ParameterOutput3 := Module[3].Output.SkillOutput[13].ParameterOutput[3];
Module[3].Input.SkillInput[13].ParameterInput[4] := Module2003.Input.SkillInput.SkillInput13.ParameterInput.ParameterInput4;
Module2003.Output.SkillOutput.SkillOutput13.ParameterOutput.ParameterOutput4 := Module[3].Output.SkillOutput[13].ParameterOutput[4];
Module[3].Input.SkillInput[13].ParameterInput[5] := Module2003.Input.SkillInput.SkillInput13.ParameterInput.ParameterInput5;
Module2003.Output.SkillOutput.SkillOutput13.ParameterOutput.ParameterOutput5 := Module[3].Output.SkillOutput[13].ParameterOutput[5];
Module[3].Input.SkillInput[14].Execute := Module2003.Input.SkillInput.SkillInput14.Execute;
Module2003.Output.SkillOutput.SkillOutput14.Dummy := Module[3].Output.SkillOutput[14].Dummy;
Module2003.Output.SkillOutput.SkillOutput14.ID := Module[3].Output.SkillOutput[14].ID;
Module2003.Output.SkillOutput.SkillOutput14.Name := Module[3].Output.SkillOutput[14].Name;
Module2003.Output.SkillOutput.SkillOutput14.Activated := Module[3].Output.SkillOutput[14].Activated;
Module2003.Output.SkillOutput.SkillOutput14.Ready := Module[3].Output.SkillOutput[14].Ready;
Module2003.Output.SkillOutput.SkillOutput14.Busy := Module[3].Output.SkillOutput[14].Busy;
Module2003.Output.SkillOutput.SkillOutput14.Done := Module[3].Output.SkillOutput[14].Done;
Module2003.Output.SkillOutput.SkillOutput14.Error := Module[3].Output.SkillOutput[14].Error;
Module2003.Output.Statevalue.Statevalue0 := Module[3].Output.Statevalue[0];
Module2003.Output.Statevalue.Statevalue1 := Module[3].Output.Statevalue[1];
Module2003.Output.Statevalue.Statevalue2 := Module[3].Output.Statevalue[2];
Module2003.Output.Statevalue.Statevalue3 := Module[3].Output.Statevalue[3];
Module2003.Output.Statevalue.Statevalue4 := Module[3].Output.Statevalue[4];
Module2003.Output.Statevalue.Statevalue5 := Module[3].Output.Statevalue[5];
Module2003.Output.Statevalue.Statevalue6 := Module[3].Output.Statevalue[6];
Module2003.Output.Statevalue.Statevalue7 := Module[3].Output.Statevalue[7];
Module2003.Output.Statevalue.Statevalue8 := Module[3].Output.Statevalue[8];
Module2003.Output.Statevalue.Statevalue9 := Module[3].Output.Statevalue[9];
Module2003.Output.Statevalue.Statevalue10 := Module[3].Output.Statevalue[10];
Module[3].Input.SkillInput[14].ParameterInput[0] := Module2003.Input.SkillInput.SkillInput14.ParameterInput.ParameterInput0;
Module2003.Output.SkillOutput.SkillOutput14.ParameterOutput.ParameterOutput0 := Module[3].Output.SkillOutput[14].ParameterOutput[0];
Module[3].Input.SkillInput[14].ParameterInput[1] := Module2003.Input.SkillInput.SkillInput14.ParameterInput.ParameterInput1;
Module2003.Output.SkillOutput.SkillOutput14.ParameterOutput.ParameterOutput1 := Module[3].Output.SkillOutput[14].ParameterOutput[1];
Module[3].Input.SkillInput[14].ParameterInput[2] := Module2003.Input.SkillInput.SkillInput14.ParameterInput.ParameterInput2;
Module2003.Output.SkillOutput.SkillOutput14.ParameterOutput.ParameterOutput2 := Module[3].Output.SkillOutput[14].ParameterOutput[2];
Module[3].Input.SkillInput[14].ParameterInput[3] := Module2003.Input.SkillInput.SkillInput14.ParameterInput.ParameterInput3;
Module2003.Output.SkillOutput.SkillOutput14.ParameterOutput.ParameterOutput3 := Module[3].Output.SkillOutput[14].ParameterOutput[3];
Module[3].Input.SkillInput[14].ParameterInput[4] := Module2003.Input.SkillInput.SkillInput14.ParameterInput.ParameterInput4;
Module2003.Output.SkillOutput.SkillOutput14.ParameterOutput.ParameterOutput4 := Module[3].Output.SkillOutput[14].ParameterOutput[4];
Module[3].Input.SkillInput[14].ParameterInput[5] := Module2003.Input.SkillInput.SkillInput14.ParameterInput.ParameterInput5;
Module2003.Output.SkillOutput.SkillOutput14.ParameterOutput.ParameterOutput5 := Module[3].Output.SkillOutput[14].ParameterOutput[5];
Module[3].Input.SkillInput[15].Execute := Module2003.Input.SkillInput.SkillInput15.Execute;
Module2003.Output.SkillOutput.SkillOutput15.Dummy := Module[3].Output.SkillOutput[15].Dummy;
Module2003.Output.SkillOutput.SkillOutput15.ID := Module[3].Output.SkillOutput[15].ID;
Module2003.Output.SkillOutput.SkillOutput15.Name := Module[3].Output.SkillOutput[15].Name;
Module2003.Output.SkillOutput.SkillOutput15.Activated := Module[3].Output.SkillOutput[15].Activated;
Module2003.Output.SkillOutput.SkillOutput15.Ready := Module[3].Output.SkillOutput[15].Ready;
Module2003.Output.SkillOutput.SkillOutput15.Busy := Module[3].Output.SkillOutput[15].Busy;
Module2003.Output.SkillOutput.SkillOutput15.Done := Module[3].Output.SkillOutput[15].Done;
Module2003.Output.SkillOutput.SkillOutput15.Error := Module[3].Output.SkillOutput[15].Error;
Module2003.Output.Statevalue.Statevalue0 := Module[3].Output.Statevalue[0];
Module2003.Output.Statevalue.Statevalue1 := Module[3].Output.Statevalue[1];
Module2003.Output.Statevalue.Statevalue2 := Module[3].Output.Statevalue[2];
Module2003.Output.Statevalue.Statevalue3 := Module[3].Output.Statevalue[3];
Module2003.Output.Statevalue.Statevalue4 := Module[3].Output.Statevalue[4];
Module2003.Output.Statevalue.Statevalue5 := Module[3].Output.Statevalue[5];
Module2003.Output.Statevalue.Statevalue6 := Module[3].Output.Statevalue[6];
Module2003.Output.Statevalue.Statevalue7 := Module[3].Output.Statevalue[7];
Module2003.Output.Statevalue.Statevalue8 := Module[3].Output.Statevalue[8];
Module2003.Output.Statevalue.Statevalue9 := Module[3].Output.Statevalue[9];
Module2003.Output.Statevalue.Statevalue10 := Module[3].Output.Statevalue[10];
Module[3].Input.SkillInput[15].ParameterInput[0] := Module2003.Input.SkillInput.SkillInput15.ParameterInput.ParameterInput0;
Module2003.Output.SkillOutput.SkillOutput15.ParameterOutput.ParameterOutput0 := Module[3].Output.SkillOutput[15].ParameterOutput[0];
Module[3].Input.SkillInput[15].ParameterInput[1] := Module2003.Input.SkillInput.SkillInput15.ParameterInput.ParameterInput1;
Module2003.Output.SkillOutput.SkillOutput15.ParameterOutput.ParameterOutput1 := Module[3].Output.SkillOutput[15].ParameterOutput[1];
Module[3].Input.SkillInput[15].ParameterInput[2] := Module2003.Input.SkillInput.SkillInput15.ParameterInput.ParameterInput2;
Module2003.Output.SkillOutput.SkillOutput15.ParameterOutput.ParameterOutput2 := Module[3].Output.SkillOutput[15].ParameterOutput[2];
Module[3].Input.SkillInput[15].ParameterInput[3] := Module2003.Input.SkillInput.SkillInput15.ParameterInput.ParameterInput3;
Module2003.Output.SkillOutput.SkillOutput15.ParameterOutput.ParameterOutput3 := Module[3].Output.SkillOutput[15].ParameterOutput[3];
Module[3].Input.SkillInput[15].ParameterInput[4] := Module2003.Input.SkillInput.SkillInput15.ParameterInput.ParameterInput4;
Module2003.Output.SkillOutput.SkillOutput15.ParameterOutput.ParameterOutput4 := Module[3].Output.SkillOutput[15].ParameterOutput[4];
Module[3].Input.SkillInput[15].ParameterInput[5] := Module2003.Input.SkillInput.SkillInput15.ParameterInput.ParameterInput5;
Module2003.Output.SkillOutput.SkillOutput15.ParameterOutput.ParameterOutput5 := Module[3].Output.SkillOutput[15].ParameterOutput[5];
END_IF

END_FUNCTION_BLOCK

// ---- POUs/SkillHandle/FB_TEST1.TcPOU
FUNCTION_BLOCK FB_TEST1
VAR_INPUT
	execute: BOOL;
END_VAR
VAR
	TIMERDONE: BOOL;
END_VAR

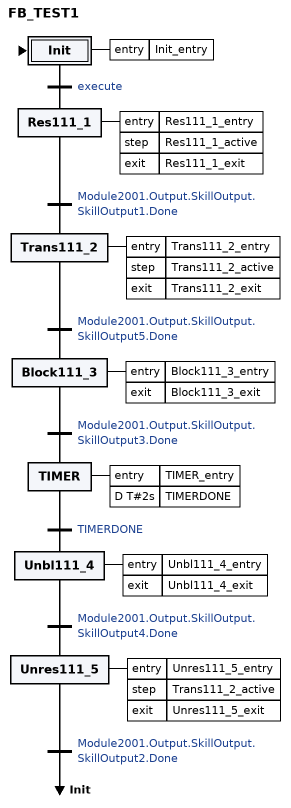
INITIAL_STEP Init:
    Init_entry(P1);  // entry action
END_STEP
TRANSITION FROM Init TO Res111_1
    := execute;
END_TRANSITION
STEP Res111_1:
    Res111_1_entry(P1);  // entry action
    Res111_1_active(N);  // step action
    Res111_1_exit(P0);  // exit action
END_STEP
TRANSITION FROM Res111_1 TO Trans111_2
    := Module2001.Output.SkillOutput.SkillOutput1.Done;
END_TRANSITION
STEP Trans111_2:
    Trans111_2_entry(P1);  // entry action
    Trans111_2_active(N);  // step action
    Trans111_2_exit(P0);  // exit action
END_STEP
TRANSITION FROM Trans111_2 TO Block111_3
    := Module2001.Output.SkillOutput.SkillOutput5.Done;
END_TRANSITION
STEP Block111_3:
    Block111_3_entry(P1);  // entry action
    Block111_3_exit(P0);  // exit action
END_STEP
TRANSITION FROM Block111_3 TO TIMER
    := Module2001.Output.SkillOutput.SkillOutput3.Done;
END_TRANSITION
STEP TIMER:
    TIMER_entry(P1);  // entry action
    TIMERDONE(D, T#2s);
END_STEP
TRANSITION FROM TIMER TO Unbl111_4
    := TIMERDONE;
END_TRANSITION
STEP Unbl111_4:
    Unbl111_4_entry(P1);  // entry action
    Unbl111_4_exit(P0);  // exit action
END_STEP
TRANSITION FROM Unbl111_4 TO Unres111_5
    := Module2001.Output.SkillOutput.SkillOutput4.Done;
END_TRANSITION
STEP Unres111_5:
    Unres111_5_entry(P1);  // entry action
    Trans111_2_active(N);  // step action
    Unres111_5_exit(P0);  // exit action
END_STEP
TRANSITION FROM Unres111_5 TO Init
    := Module2001.Output.SkillOutput.SkillOutput2.Done;
END_TRANSITION

ACTION Block111_3_entry:
//BLOCKIEREN

Module2001.Input.SkillInput.SkillInput3.Execute := TRUE;
Module2001.Input.SkillInput.SkillInput3.ParameterInput.Parameterinput1.Value := 111; //TaskID
END_ACTION

ACTION Res111_1_exit:
// Reservieren entry
Module2001.Input.SkillInput.SkillInput1.Execute := FALSE;
Module2001.Input.SkillInput.SkillInput1.ParameterInput.Parameterinput1.Value := 0; //TASKID
END_ACTION

ACTION Trans111_2_exit:
//TRANSPORTIEREN

Module2001.Input.SkillInput.SkillInput5.Execute := FALSE;
Module2001.Input.SkillInput.SkillInput5.ParameterInput.Parameterinput1.Value := 0; //X-Position
Module2001.Input.SkillInput.SkillInput5.ParameterInput.Parameterinput2.Value := 0; //Z-Position
Module2001.Input.SkillInput.SkillInput5.ParameterInput.Parameterinput3.Value := 0; //Velocity
Module2001.Input.SkillInput.SkillInput5.ParameterInput.Parameterinput4.Value := 0; //Acceleration
END_ACTION

ACTION Res111_1_entry:
// Reservieren entry
Module2001.Input.SkillInput.SkillInput1.Execute := TRUE;
Module2001.Input.SkillInput.SkillInput1.ParameterInput.Parameterinput1.Value := 111; //TASKID
END_ACTION

ACTION Unres111_5_exit:
//unreserve
Module2001.Input.SkillInput.SkillInput2.Execute := FALSE;
Module2001.Input.SkillInput.SkillInput2.ParameterInput.Parameterinput1.Value := 0; //TaskID
END_ACTION

ACTION Unbl111_4_entry:
//unBLOCKIEREN

Module2001.Input.SkillInput.SkillInput4.Execute := TRUE; //FALSE weil timer
Module2001.Input.SkillInput.SkillInput4.ParameterInput.Parameterinput1.Value := 111; //TaskID
END_ACTION

ACTION Block111_3_exit:
//BLOCKIEREN

Module2001.Input.SkillInput.SkillInput3.Execute := FALSE;
Module2001.Input.SkillInput.SkillInput3.ParameterInput.Parameterinput1.Value := 0; //TaskID
END_ACTION

ACTION Init_entry:
execute := FALSE;
END_ACTION

ACTION Res111_1_active:

END_ACTION

ACTION Unres111_5_entry:
//unreserve
Module2001.Input.SkillInput.SkillInput2.Execute := TRUE;
Module2001.Input.SkillInput.SkillInput2.ParameterInput.Parameterinput1.Value := 111; //TaskID
END_ACTION

ACTION Unbl111_4_exit:
//unBLOCKIEREN

Module2001.Input.SkillInput.SkillInput4.Execute := FALSE; 
Module2001.Input.SkillInput.SkillInput4.ParameterInput.Parameterinput1.Value := 000; //TaskID
END_ACTION

ACTION TIMER_entry:
TIMERDONE := FALSE;
END_ACTION

ACTION Trans111_2_active:

END_ACTION

ACTION Trans111_2_entry:
//TRANSPORTIEREN

Module2001.Input.SkillInput.SkillInput5.Execute := TRUE;
Module2001.Input.SkillInput.SkillInput5.ParameterInput.Parameterinput1.Value := 3450; //X-Position
Module2001.Input.SkillInput.SkillInput5.ParameterInput.Parameterinput2.Value := 0;//90; //Z-Position
Module2001.Input.SkillInput.SkillInput5.ParameterInput.Parameterinput3.Value := 300; //Velocity
Module2001.Input.SkillInput.SkillInput5.ParameterInput.Parameterinput4.Value := 0; //Acceleration
END_ACTION

END_FUNCTION_BLOCK

// ---- POUs/SkillHandle/FB_TEST2.TcPOU
FUNCTION_BLOCK FB_TEST2
VAR_INPUT
	execute: BOOL;
	pos2: LREAL := 2500;
END_VAR
VAR
	TIMERDONE: BOOL;
END_VAR

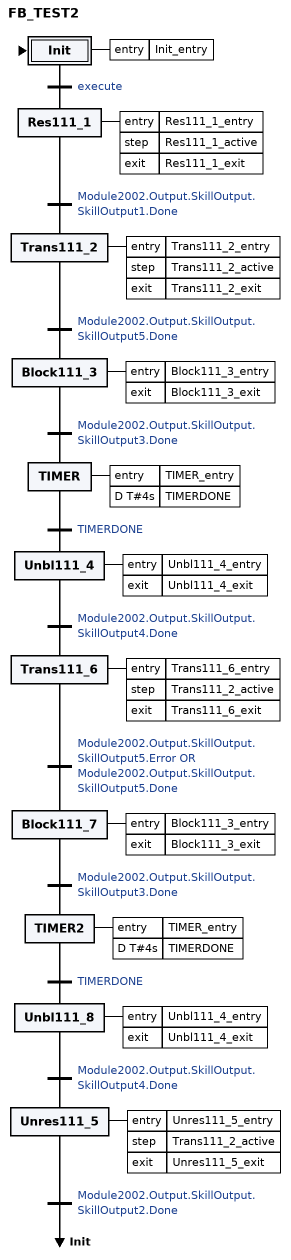
INITIAL_STEP Init:
    Init_entry(P1);  // entry action
END_STEP
TRANSITION FROM Init TO Res111_1
    := execute;
END_TRANSITION
STEP Res111_1:
    Res111_1_entry(P1);  // entry action
    Res111_1_active(N);  // step action
    Res111_1_exit(P0);  // exit action
END_STEP
TRANSITION FROM Res111_1 TO Trans111_2
    := Module2002.Output.SkillOutput.SkillOutput1.Done;
END_TRANSITION
STEP Trans111_2:
    Trans111_2_entry(P1);  // entry action
    Trans111_2_active(N);  // step action
    Trans111_2_exit(P0);  // exit action
END_STEP
TRANSITION FROM Trans111_2 TO Block111_3
    := Module2002.Output.SkillOutput.SkillOutput5.Done;
END_TRANSITION
STEP Block111_3:
    Block111_3_entry(P1);  // entry action
    Block111_3_exit(P0);  // exit action
END_STEP
TRANSITION FROM Block111_3 TO TIMER
    := Module2002.Output.SkillOutput.SkillOutput3.Done;
END_TRANSITION
STEP TIMER:
    TIMER_entry(P1);  // entry action
    TIMERDONE(D, T#4s);
END_STEP
TRANSITION FROM TIMER TO Unbl111_4
    := TIMERDONE;
END_TRANSITION
STEP Unbl111_4:
    Unbl111_4_entry(P1);  // entry action
    Unbl111_4_exit(P0);  // exit action
END_STEP
TRANSITION FROM Unbl111_4 TO Trans111_6
    := Module2002.Output.SkillOutput.SkillOutput4.Done;
END_TRANSITION
STEP Trans111_6:
    Trans111_6_entry(P1);  // entry action
    Trans111_2_active(N);  // step action
    Trans111_6_exit(P0);  // exit action
END_STEP
TRANSITION FROM Trans111_6 TO Block111_7
    := Module2002.Output.SkillOutput.SkillOutput5.Error OR Module2002.Output.SkillOutput.SkillOutput5.Done;
END_TRANSITION
STEP Block111_7:
    Block111_3_entry(P1);  // entry action
    Block111_3_exit(P0);  // exit action
END_STEP
TRANSITION FROM Block111_7 TO TIMER2
    := Module2002.Output.SkillOutput.SkillOutput3.Done;
END_TRANSITION
STEP TIMER2:
    TIMER_entry(P1);  // entry action
    TIMERDONE(D, T#4s);
END_STEP
TRANSITION FROM TIMER2 TO Unbl111_8
    := TIMERDONE;
END_TRANSITION
STEP Unbl111_8:
    Unbl111_4_entry(P1);  // entry action
    Unbl111_4_exit(P0);  // exit action
END_STEP
TRANSITION FROM Unbl111_8 TO Unres111_5
    := Module2002.Output.SkillOutput.SkillOutput4.Done;
END_TRANSITION
STEP Unres111_5:
    Unres111_5_entry(P1);  // entry action
    Trans111_2_active(N);  // step action
    Unres111_5_exit(P0);  // exit action
END_STEP
TRANSITION FROM Unres111_5 TO Init
    := Module2002.Output.SkillOutput.SkillOutput2.Done;
END_TRANSITION

ACTION Trans111_6_exit:
//TRANSPORTIEREN

Module2002.Input.SkillInput.SkillInput5.Execute := FALSE;
Module2002.Input.SkillInput.SkillInput5.ParameterInput.Parameterinput1.Value := 0; //X-Position
Module2002.Input.SkillInput.SkillInput5.ParameterInput.Parameterinput2.Value := 0; //Z-Position
Module2002.Input.SkillInput.SkillInput5.ParameterInput.Parameterinput3.Value := 0; //Velocity
Module2002.Input.SkillInput.SkillInput5.ParameterInput.Parameterinput4.Value := 0; //Acceleration
END_ACTION

ACTION Block111_3_entry:
//BLOCKIEREN

Module2002.Input.SkillInput.SkillInput3.Execute := TRUE;
Module2002.Input.SkillInput.SkillInput3.ParameterInput.Parameterinput1.Value := 112; //TaskID
END_ACTION

ACTION Trans111_6_entry:
//TRANSPORTIEREN

Module2002.Input.SkillInput.SkillInput5.Execute := TRUE;
Module2002.Input.SkillInput.SkillInput5.ParameterInput.Parameterinput1.Value := pos2; //X-Position
Module2002.Input.SkillInput.SkillInput5.ParameterInput.Parameterinput2.Value := 80; //Z-Position
Module2002.Input.SkillInput.SkillInput5.ParameterInput.Parameterinput3.Value := 0; //Velocity
Module2002.Input.SkillInput.SkillInput5.ParameterInput.Parameterinput4.Value := 0; //Acceleration
END_ACTION

ACTION Init_entry:
execute := FALSE;
END_ACTION

ACTION Trans111_2_entry:
//TRANSPORTIEREN

Module2002.Input.SkillInput.SkillInput5.Execute := TRUE;
Module2002.Input.SkillInput.SkillInput5.ParameterInput.Parameterinput1.Value := 3000; //X-Position
Module2002.Input.SkillInput.SkillInput5.ParameterInput.Parameterinput2.Value := 0; //Z-Position
Module2002.Input.SkillInput.SkillInput5.ParameterInput.Parameterinput3.Value := 0; //Velocity
Module2002.Input.SkillInput.SkillInput5.ParameterInput.Parameterinput4.Value := 0; //Acceleration
END_ACTION

ACTION Res111_1_entry:
// Reservieren entry
Module2002.Input.SkillInput.SkillInput1.Execute := TRUE;
Module2002.Input.SkillInput.SkillInput1.ParameterInput.Parameterinput1.Value := 112; //TASKID
END_ACTION

ACTION Unbl111_4_exit:
//unBLOCKIEREN

Module2002.Input.SkillInput.SkillInput4.Execute := FALSE; 
Module2002.Input.SkillInput.SkillInput4.ParameterInput.Parameterinput1.Value := 000; //TaskID
END_ACTION

ACTION Unres111_5_entry:
//unreserve
Module2002.Input.SkillInput.SkillInput2.Execute := TRUE;
Module2002.Input.SkillInput.SkillInput2.ParameterInput.Parameterinput1.Value := 112; //TaskID
END_ACTION

ACTION Res111_1_active:

END_ACTION

ACTION Trans111_2_exit:
//TRANSPORTIEREN

Module2002.Input.SkillInput.SkillInput5.Execute := FALSE;
Module2002.Input.SkillInput.SkillInput5.ParameterInput.Parameterinput1.Value := 0; //X-Position
Module2002.Input.SkillInput.SkillInput5.ParameterInput.Parameterinput2.Value := 0; //Z-Position
Module2002.Input.SkillInput.SkillInput5.ParameterInput.Parameterinput3.Value := 0; //Velocity
Module2002.Input.SkillInput.SkillInput5.ParameterInput.Parameterinput4.Value := 0; //Acceleration
END_ACTION

ACTION TIMER_entry:
TIMERDONE := FALSE;
END_ACTION

ACTION Trans111_2_active:

END_ACTION

ACTION Unbl111_4_entry:
//unBLOCKIEREN

Module2002.Input.SkillInput.SkillInput4.Execute := TRUE; //FALSE weil timer
Module2002.Input.SkillInput.SkillInput4.ParameterInput.Parameterinput1.Value := 112; //TaskID
END_ACTION

ACTION Trans111_2_entry_1:
//TRANSPORTIEREN

Module2002.Input.SkillInput.SkillInput5.Execute := TRUE;
Module2002.Input.SkillInput.SkillInput5.ParameterInput.Parameterinput1.Value := 3000; //X-Position
Module2002.Input.SkillInput.SkillInput5.ParameterInput.Parameterinput2.Value := 0; //Z-Position
Module2002.Input.SkillInput.SkillInput5.ParameterInput.Parameterinput3.Value := 0; //Velocity
Module2002.Input.SkillInput.SkillInput5.ParameterInput.Parameterinput4.Value := 0; //Acceleration
END_ACTION

ACTION Unres111_5_exit:
//unreserve
Module2002.Input.SkillInput.SkillInput2.Execute := FALSE;
Module2002.Input.SkillInput.SkillInput2.ParameterInput.Parameterinput1.Value := 0; //TaskID
END_ACTION

ACTION Block111_3_exit:
//BLOCKIEREN

Module2002.Input.SkillInput.SkillInput3.Execute := FALSE;
Module2002.Input.SkillInput.SkillInput3.ParameterInput.Parameterinput1.Value := 0; //TaskID
END_ACTION

ACTION Res111_1_exit:
// Reservieren entry
Module2002.Input.SkillInput.SkillInput1.Execute := FALSE;
Module2002.Input.SkillInput.SkillInput1.ParameterInput.Parameterinput1.Value := 0; //TASKID
END_ACTION

END_FUNCTION_BLOCK

// ---- POUs/SkillHandle/FB_TEST3.TcPOU
FUNCTION_BLOCK FB_TEST3
VAR_INPUT
	execute: BOOL;
	pos2: LREAL := 2500;
END_VAR
VAR
	TIMERDONE: BOOL;
END_VAR

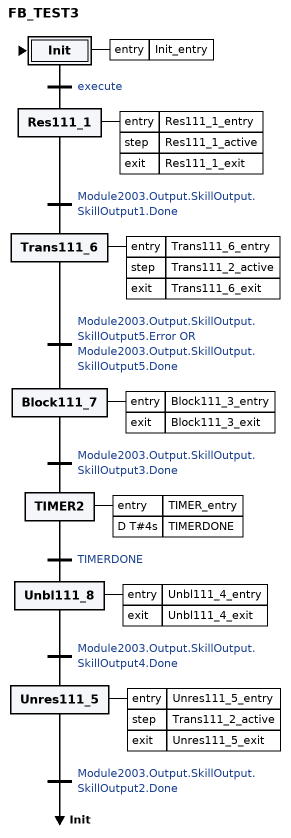
INITIAL_STEP Init:
    Init_entry(P1);  // entry action
END_STEP
TRANSITION FROM Init TO Res111_1
    := execute;
END_TRANSITION
STEP Res111_1:
    Res111_1_entry(P1);  // entry action
    Res111_1_active(N);  // step action
    Res111_1_exit(P0);  // exit action
END_STEP
TRANSITION FROM Res111_1 TO Trans111_6
    := Module2003.Output.SkillOutput.SkillOutput1.Done;
END_TRANSITION
STEP Trans111_6:
    Trans111_6_entry(P1);  // entry action
    Trans111_2_active(N);  // step action
    Trans111_6_exit(P0);  // exit action
END_STEP
TRANSITION FROM Trans111_6 TO Block111_7
    := Module2003.Output.SkillOutput.SkillOutput5.Error OR Module2003.Output.SkillOutput.SkillOutput5.Done;
END_TRANSITION
STEP Block111_7:
    Block111_3_entry(P1);  // entry action
    Block111_3_exit(P0);  // exit action
END_STEP
TRANSITION FROM Block111_7 TO TIMER2
    := Module2003.Output.SkillOutput.SkillOutput3.Done;
END_TRANSITION
STEP TIMER2:
    TIMER_entry(P1);  // entry action
    TIMERDONE(D, T#4s);
END_STEP
TRANSITION FROM TIMER2 TO Unbl111_8
    := TIMERDONE;
END_TRANSITION
STEP Unbl111_8:
    Unbl111_4_entry(P1);  // entry action
    Unbl111_4_exit(P0);  // exit action
END_STEP
TRANSITION FROM Unbl111_8 TO Unres111_5
    := Module2003.Output.SkillOutput.SkillOutput4.Done;
END_TRANSITION
STEP Unres111_5:
    Unres111_5_entry(P1);  // entry action
    Trans111_2_active(N);  // step action
    Unres111_5_exit(P0);  // exit action
END_STEP
TRANSITION FROM Unres111_5 TO Init
    := Module2003.Output.SkillOutput.SkillOutput2.Done;
END_TRANSITION

ACTION Trans111_6_exit:
//TRANSPORTIEREN

Module2003.Input.SkillInput.SkillInput5.Execute := FALSE;
Module2003.Input.SkillInput.SkillInput5.ParameterInput.Parameterinput1.Value := 0; //X-Position
Module2003.Input.SkillInput.SkillInput5.ParameterInput.Parameterinput2.Value := 0; //Z-Position
Module2003.Input.SkillInput.SkillInput5.ParameterInput.Parameterinput3.Value := 0; //Velocity
Module2003.Input.SkillInput.SkillInput5.ParameterInput.Parameterinput4.Value := 0; //Acceleration
END_ACTION

ACTION Res111_1_entry:
// Reservieren entry
Module2003.Input.SkillInput.SkillInput1.Execute := TRUE;
Module2003.Input.SkillInput.SkillInput1.ParameterInput.Parameterinput1.Value := 113; //TASKID
END_ACTION

ACTION Res111_1_active:

END_ACTION

ACTION Res111_1_exit:
// Reservieren entry
Module2003.Input.SkillInput.SkillInput1.Execute := FALSE;
Module2003.Input.SkillInput.SkillInput1.ParameterInput.Parameterinput1.Value := 0; //TASKID
END_ACTION

ACTION TIMER_entry:
TIMERDONE := FALSE;
END_ACTION

ACTION Trans111_6_entry:
//TRANSPORTIEREN

Module2003.Input.SkillInput.SkillInput5.Execute := TRUE;
Module2003.Input.SkillInput.SkillInput5.ParameterInput.Parameterinput1.Value := 2800; //X-Position
Module2003.Input.SkillInput.SkillInput5.ParameterInput.Parameterinput2.Value := 80; //Z-Position
Module2003.Input.SkillInput.SkillInput5.ParameterInput.Parameterinput3.Value := 0; //Velocity
Module2003.Input.SkillInput.SkillInput5.ParameterInput.Parameterinput4.Value := 0; //Acceleration
END_ACTION

ACTION Unbl111_4_exit:
//unBLOCKIEREN

Module2003.Input.SkillInput.SkillInput4.Execute := FALSE; 
Module2003.Input.SkillInput.SkillInput4.ParameterInput.Parameterinput1.Value := 000; //TaskID
END_ACTION

ACTION Trans111_2_entry:
//TRANSPORTIEREN

Module2003.Input.SkillInput.SkillInput5.Execute := TRUE;
Module2003.Input.SkillInput.SkillInput5.ParameterInput.Parameterinput1.Value := 2400; //X-Position
Module2003.Input.SkillInput.SkillInput5.ParameterInput.Parameterinput2.Value := 0; //Z-Position
Module2003.Input.SkillInput.SkillInput5.ParameterInput.Parameterinput3.Value := 300; //Velocity
Module2003.Input.SkillInput.SkillInput5.ParameterInput.Parameterinput4.Value := 100; //Acceleration
END_ACTION

ACTION Trans111_2_active:

END_ACTION

ACTION Unres111_5_exit:
//unreserve
Module2003.Input.SkillInput.SkillInput2.Execute := FALSE;
Module2003.Input.SkillInput.SkillInput2.ParameterInput.Parameterinput1.Value := 0; //TaskID
END_ACTION

ACTION Init_entry:
execute := FALSE;
END_ACTION

ACTION Trans111_2_exit:
//TRANSPORTIEREN

Module2003.Input.SkillInput.SkillInput5.Execute := FALSE;
Module2003.Input.SkillInput.SkillInput5.ParameterInput.Parameterinput1.Value := 0; //X-Position
Module2003.Input.SkillInput.SkillInput5.ParameterInput.Parameterinput2.Value := 0; //Z-Position
Module2003.Input.SkillInput.SkillInput5.ParameterInput.Parameterinput3.Value := 0; //Velocity
Module2003.Input.SkillInput.SkillInput5.ParameterInput.Parameterinput4.Value := 0; //Acceleration
END_ACTION

ACTION Block111_3_entry:
//BLOCKIEREN

Module2003.Input.SkillInput.SkillInput3.Execute := TRUE;
Module2003.Input.SkillInput.SkillInput3.ParameterInput.Parameterinput1.Value := 113; //TaskID
END_ACTION

ACTION Unres111_5_entry:
//unreserve
Module2003.Input.SkillInput.SkillInput2.Execute := TRUE;
Module2003.Input.SkillInput.SkillInput2.ParameterInput.Parameterinput1.Value := 113; //TaskID
END_ACTION

ACTION Block111_3_exit:
//BLOCKIEREN

Module2003.Input.SkillInput.SkillInput3.Execute := FALSE;
Module2003.Input.SkillInput.SkillInput3.ParameterInput.Parameterinput1.Value := 0; //TaskID
END_ACTION

ACTION Unbl111_4_entry:
//unBLOCKIEREN

Module2003.Input.SkillInput.SkillInput4.Execute := TRUE; //FALSE weil timer
Module2003.Input.SkillInput.SkillInput4.ParameterInput.Parameterinput1.Value := 112; //TaskID
END_ACTION

END_FUNCTION_BLOCK

// ---- POUs/SkillHandle/Fb_Test_init_x.TcPOU
FUNCTION_BLOCK Fb_Test_init_x
VAR_INPUT
	execute: BOOL;
END_VAR

IF execute  THEN
	MI5.Module2001.Input.SkillInput.SkillInput0.ParameterInput.ParameterInput0.StringValue := 'opc.tcp://192.168.192.117:4840';
	MI5.Module2001.Input.SkillInput.SkillInput0.ParameterInput.ParameterInput1.StringValue := 'MI5.Module1202.Output.PositionSensor';
	MI5.Module2001.Input.SkillInput.SkillInput0.ParameterInput.ParameterInput2.StringValue := 'MI5.Module1202.Input.PositionInput';
	MI5.Module2001.Input.SkillInput.SkillInput0.ParameterInput.ParameterInput3.StringValue := '4';
	MI5.Module2001.Input.SkillInput.SkillInput0.ParameterInput.ParameterInput4.StringValue := 'PLC1';
	MI5.Module2001.Input.SkillInput.SkillInput0.Execute := TRUE;
	IF MI5.Module2001.Output.SkillOutput.SkillOutput0.Done OR MI5.Module2001.Output.SkillOutput.SkillOutput0.Error THEN
		MI5.Module2001.Input.SkillInput.SkillInput0.Execute := FALSE;
		execute := FALSE;
	END_IF
END_IF

END_FUNCTION_BLOCK

// ---- POUs/SkillHandle/Fb_Test_init_y.TcPOU
FUNCTION_BLOCK Fb_Test_init_y
VAR_INPUT
	execute: BOOL;
END_VAR

IF execute  THEN
	MI5.Module2001.Input.SkillInput.SkillInput0.ParameterInput.ParameterInput0.StringValue := 'opc.tcp://192.168.192.118:4840';
	MI5.Module2001.Input.SkillInput.SkillInput0.ParameterInput.ParameterInput1.StringValue := 'MI5.Module1203.Output.PositionSensor';
	MI5.Module2001.Input.SkillInput.SkillInput0.ParameterInput.ParameterInput2.StringValue := 'MI5.Module1203.Input.PositionInput';
	MI5.Module2001.Input.SkillInput.SkillInput0.ParameterInput.ParameterInput3.StringValue := '4';
	MI5.Module2001.Input.SkillInput.SkillInput0.ParameterInput.ParameterInput4.StringValue := 'PLC1';
	MI5.Module2001.Input.SkillInput.SkillInput0.Execute := TRUE;
	IF MI5.Module2001.Output.SkillOutput.SkillOutput0.Done OR MI5.Module2001.Output.SkillOutput.SkillOutput0.Error THEN
		MI5.Module2001.Input.SkillInput.SkillInput0.Execute := FALSE;
		execute := FALSE;
	END_IF
END_IF

END_FUNCTION_BLOCK

// ---- POUs/SkillHandle/Fb_Test_init_z.TcPOU
FUNCTION_BLOCK Fb_Test_init_z
VAR_INPUT
	execute: BOOL;
END_VAR

IF execute THEN
	MI5.Module2001.Input.SkillInput.SkillInput0.ParameterInput.ParameterInput0.StringValue := 'opc.tcp://192.168.192.119:4840';
	MI5.Module2001.Input.SkillInput.SkillInput0.ParameterInput.ParameterInput1.StringValue := 'MI5.Module1204.Output.PositionSensor';
	MI5.Module2001.Input.SkillInput.SkillInput0.ParameterInput.ParameterInput2.StringValue := 'MI5.Module1204.Input.PositionInput';
	MI5.Module2001.Input.SkillInput.SkillInput0.ParameterInput.ParameterInput3.StringValue := '4';
	MI5.Module2001.Input.SkillInput.SkillInput0.ParameterInput.ParameterInput4.StringValue := 'PLC1';
	MI5.Module2001.Input.SkillInput.SkillInput0.Execute := TRUE;
	IF MI5.Module2001.Output.SkillOutput.SkillOutput0.Done OR MI5.Module2001.Output.SkillOutput.SkillOutput0.Error THEN
		MI5.Module2001.Input.SkillInput.SkillInput0.Execute := FALSE;
		execute := FALSE;
	END_IF
END_IF

END_FUNCTION_BLOCK

// ---- POUs/SkillHandle/FB_ResetXTS.TcPOU
FUNCTION_BLOCK FB_ResetXTS
VAR_INPUT
	execute: BOOL;
END_VAR
VAR
	state: INT := 0;
	i: INT;
	cyclecnt: INT := 0;
	skillcyclecnt: INT := 0;
	processcycles: INT := 5;
END_VAR

IF execute THEN
	CASE state OF
	-1: 
		skillcyclecnt 	:= 0;
		cyclecnt		:= 0;
		state := 0;
	0:
		MI5.Module2001.Input.SkillInput.SkillInput0.Execute := FALSE;	
		MI5.Module2001.Input.SkillInput.SkillInput1.Execute := FALSE;
		MI5.Module2001.Input.SkillInput.SkillInput2.Execute := TRUE;
		MI5.Module2001.Input.SkillInput.SkillInput3.Execute := FALSE;
		MI5.Module2001.Input.SkillInput.SkillInput4.Execute := TRUE;
		MI5.Module2001.Input.SkillInput.SkillInput5.Execute := FALSE;
		
		MI5.Module2002.Input.SkillInput.SkillInput0.Execute := FALSE;	
		MI5.Module2002.Input.SkillInput.SkillInput1.Execute := FALSE;
		MI5.Module2002.Input.SkillInput.SkillInput2.Execute := TRUE;
		MI5.Module2002.Input.SkillInput.SkillInput3.Execute := FALSE;
		MI5.Module2002.Input.SkillInput.SkillInput4.Execute := TRUE;
		MI5.Module2002.Input.SkillInput.SkillInput5.Execute := FALSE;
		
		MI5.Module2003.Input.SkillInput.SkillInput0.Execute := FALSE;	
		MI5.Module2003.Input.SkillInput.SkillInput1.Execute := FALSE;
		MI5.Module2003.Input.SkillInput.SkillInput2.Execute := TRUE;
		MI5.Module2003.Input.SkillInput.SkillInput3.Execute := FALSE;
		MI5.Module2003.Input.SkillInput.SkillInput4.Execute := TRUE;
		MI5.Module2003.Input.SkillInput.SkillInput5.Execute := FALSE;
		cyclecnt := cyclecnt +1;
		IF cyclecnt > processcycles THEN
			state := 10;
			cyclecnt := 0;
		END_IF
	
	10: 
		MI5.Module2001.Input.SkillInput.SkillInput0.Execute := FALSE;	
		MI5.Module2001.Input.SkillInput.SkillInput1.Execute := FALSE;
		MI5.Module2001.Input.SkillInput.SkillInput2.Execute := FALSE;
		MI5.Module2001.Input.SkillInput.SkillInput3.Execute := FALSE;
		MI5.Module2001.Input.SkillInput.SkillInput4.Execute := FALSE;
		MI5.Module2001.Input.SkillInput.SkillInput5.Execute := FALSE;
		
		MI5.Module2002.Input.SkillInput.SkillInput0.Execute := FALSE;	
		MI5.Module2002.Input.SkillInput.SkillInput1.Execute := FALSE;
		MI5.Module2002.Input.SkillInput.SkillInput2.Execute := FALSE;
		MI5.Module2002.Input.SkillInput.SkillInput3.Execute := FALSE;
		MI5.Module2002.Input.SkillInput.SkillInput4.Execute := FALSE;
		MI5.Module2002.Input.SkillInput.SkillInput5.Execute := FALSE;
		
		MI5.Module2003.Input.SkillInput.SkillInput0.Execute := FALSE;	
		MI5.Module2003.Input.SkillInput.SkillInput1.Execute := FALSE;
		MI5.Module2003.Input.SkillInput.SkillInput2.Execute := FALSE;
		MI5.Module2003.Input.SkillInput.SkillInput3.Execute := FALSE;
		MI5.Module2003.Input.SkillInput.SkillInput4.Execute := FALSE;
		MI5.Module2003.Input.SkillInput.SkillInput5.Execute := FALSE;
		cyclecnt := cyclecnt +1;
		IF cyclecnt > processcycles THEN
			
			cyclecnt := 0;
			skillcyclecnt := skillcyclecnt +1;
			IF skillcyclecnt > processcycles THEN
				state := 15;
				skillcyclecnt := 0;
			ELSE
				state := 0;
			END_IF
		END_IF
	15: state := 20;
		FOR i := 1 TO grpcnt DO
			IF Moverinfo[i].reserved OR MoverInfo[i].blocked THEN
				state := -1;				
			END_IF
		END_FOR
	
	20:	mi5.ResetXTS := FALSE;
		state := 0;
		execute := FALSE;
		
	
	
	
	
	END_CASE
END_IF

END_FUNCTION_BLOCK

// ---- POUs/SkillHandle/Fb_Test_init_Creme1.TcPOU
FUNCTION_BLOCK Fb_Test_init_Creme1
VAR_INPUT
	execute: BOOL;
END_VAR

IF execute THEN
	MI5.Module2001.Input.SkillInput.SkillInput0.ParameterInput.ParameterInput0.StringValue := 'opc.tcp://192.168.192.138:4840';
	MI5.Module2001.Input.SkillInput.SkillInput0.ParameterInput.ParameterInput1.StringValue := 'MI5.Module2301.Output.PositionSensor';
	MI5.Module2001.Input.SkillInput.SkillInput0.ParameterInput.ParameterInput2.StringValue := 'MI5.Module2301.Input.PositionInput';
	MI5.Module2001.Input.SkillInput.SkillInput0.ParameterInput.ParameterInput3.StringValue := '4';
	MI5.Module2001.Input.SkillInput.SkillInput0.ParameterInput.ParameterInput4.StringValue := 'PLC1';
	MI5.Module2001.Input.SkillInput.SkillInput0.Execute := TRUE;
	IF MI5.Module2001.Output.SkillOutput.SkillOutput0.Done OR MI5.Module2001.Output.SkillOutput.SkillOutput0.Error THEN
		MI5.Module2001.Input.SkillInput.SkillInput0.Execute := FALSE;
		execute := FALSE;
	END_IF
END_IF

END_FUNCTION_BLOCK

// ---- POUs/SkillHandle/Fb_Test_init_Cocktail.TcPOU
FUNCTION_BLOCK Fb_Test_init_Cocktail
VAR_INPUT
	execute: BOOL;
END_VAR

IF execute THEN
	MI5.Module2001.Input.SkillInput.SkillInput0.ParameterInput.ParameterInput0.StringValue := 'opc.tcp://192.168.192.121:4840';
	MI5.Module2001.Input.SkillInput.SkillInput0.ParameterInput.ParameterInput1.StringValue := '::AsGlobalPV:Module2201.Output.PositionSensor';
	MI5.Module2001.Input.SkillInput.SkillInput0.ParameterInput.ParameterInput2.StringValue := '::AsGlobalPV:Module2201.Input.PositionInput';
	MI5.Module2001.Input.SkillInput.SkillInput0.ParameterInput.ParameterInput3.StringValue := '6';
	MI5.Module2001.Input.SkillInput.SkillInput0.ParameterInput.ParameterInput4.StringValue := 'urn:B&R/plc/';
	MI5.Module2001.Input.SkillInput.SkillInput0.Execute := TRUE;
	IF MI5.Module2001.Output.SkillOutput.SkillOutput0.Done OR MI5.Module2001.Output.SkillOutput.SkillOutput0.Error THEN
		MI5.Module2001.Input.SkillInput.SkillInput0.Execute := FALSE;
		execute := FALSE;
	END_IF
END_IF

END_FUNCTION_BLOCK

// ---- POUs/SkillHandle/Fb_Test_init_Cookie.TcPOU
FUNCTION_BLOCK Fb_Test_init_Cookie
VAR_INPUT
	execute: BOOL;
END_VAR

IF execute THEN
	MI5.Module2001.Input.SkillInput.SkillInput0.ParameterInput.ParameterInput0.StringValue := 'opc.tcp://192.168.192.136:4840';
	MI5.Module2001.Input.SkillInput.SkillInput0.ParameterInput.ParameterInput1.StringValue := 'MI5.Module2101.Output.PositionSensor';
	MI5.Module2001.Input.SkillInput.SkillInput0.ParameterInput.ParameterInput2.StringValue := 'MI5.Module2101.Input.PositionInput';
	MI5.Module2001.Input.SkillInput.SkillInput0.ParameterInput.ParameterInput3.StringValue := '4';
	MI5.Module2001.Input.SkillInput.SkillInput0.ParameterInput.ParameterInput4.StringValue := 'PLC1';
	MI5.Module2001.Input.SkillInput.SkillInput0.Execute := TRUE;
	IF MI5.Module2001.Output.SkillOutput.SkillOutput0.Done OR MI5.Module2001.Output.SkillOutput.SkillOutput0.Error THEN
		MI5.Module2001.Input.SkillInput.SkillInput0.Execute := FALSE;
		execute := FALSE;
	END_IF
END_IF

END_FUNCTION_BLOCK

// ---- POUs/SkillHandle/FB_SHortTEST1.TcPOU
FUNCTION_BLOCK FB_SHortTEST1
VAR_INPUT
	execute: BOOL;
END_VAR
VAR
	TIMERDONE: BOOL;
END_VAR

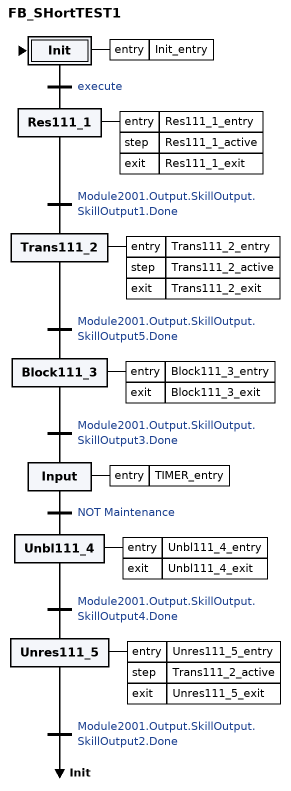
INITIAL_STEP Init:
    Init_entry(P1);  // entry action
END_STEP
TRANSITION FROM Init TO Res111_1
    := execute;
END_TRANSITION
STEP Res111_1:
    Res111_1_entry(P1);  // entry action
    Res111_1_active(N);  // step action
    Res111_1_exit(P0);  // exit action
END_STEP
TRANSITION FROM Res111_1 TO Trans111_2
    := Module2001.Output.SkillOutput.SkillOutput1.Done;
END_TRANSITION
STEP Trans111_2:
    Trans111_2_entry(P1);  // entry action
    Trans111_2_active(N);  // step action
    Trans111_2_exit(P0);  // exit action
END_STEP
TRANSITION FROM Trans111_2 TO Block111_3
    := Module2001.Output.SkillOutput.SkillOutput5.Done;
END_TRANSITION
STEP Block111_3:
    Block111_3_entry(P1);  // entry action
    Block111_3_exit(P0);  // exit action
END_STEP
TRANSITION FROM Block111_3 TO Input
    := Module2001.Output.SkillOutput.SkillOutput3.Done;
END_TRANSITION
STEP Input:
    TIMER_entry(P1);  // entry action
END_STEP
TRANSITION FROM Input TO Unbl111_4
    := NOT Maintenance;
END_TRANSITION
STEP Unbl111_4:
    Unbl111_4_entry(P1);  // entry action
    Unbl111_4_exit(P0);  // exit action
END_STEP
TRANSITION FROM Unbl111_4 TO Unres111_5
    := Module2001.Output.SkillOutput.SkillOutput4.Done;
END_TRANSITION
STEP Unres111_5:
    Unres111_5_entry(P1);  // entry action
    Trans111_2_active(N);  // step action
    Unres111_5_exit(P0);  // exit action
END_STEP
TRANSITION FROM Unres111_5 TO Init
    := Module2001.Output.SkillOutput.SkillOutput2.Done;
END_TRANSITION

ACTION Res111_1_active:

END_ACTION

ACTION Res111_1_entry:
// Reservieren entry
Module2001.Input.SkillInput.SkillInput1.Execute := TRUE;
Module2001.Input.SkillInput.SkillInput1.ParameterInput.Parameterinput1.Value := 111; //TASKID
END_ACTION

ACTION Block111_3_exit:
//BLOCKIEREN

Module2001.Input.SkillInput.SkillInput3.Execute := FALSE;
Module2001.Input.SkillInput.SkillInput3.ParameterInput.Parameterinput1.Value := 0; //TaskID
END_ACTION

ACTION Unbl111_4_entry:
//unBLOCKIEREN

Module2001.Input.SkillInput.SkillInput4.Execute := TRUE; //FALSE weil timer
Module2001.Input.SkillInput.SkillInput4.ParameterInput.Parameterinput1.Value := 111; //TaskID
END_ACTION

ACTION Trans111_2_entry:
//TRANSPORTIEREN

Module2001.Input.SkillInput.SkillInput5.Execute := TRUE;
Module2001.Input.SkillInput.SkillInput5.ParameterInput.Parameterinput1.Value := 3450; //X-Position
Module2001.Input.SkillInput.SkillInput5.ParameterInput.Parameterinput2.Value := 105;//90; //Z-Position
Module2001.Input.SkillInput.SkillInput5.ParameterInput.Parameterinput3.Value := 400; //Velocity
Module2001.Input.SkillInput.SkillInput5.ParameterInput.Parameterinput4.Value := 0; //Acceleration
END_ACTION

ACTION Block111_3_entry:
//BLOCKIEREN

Module2001.Input.SkillInput.SkillInput3.Execute := TRUE;
Module2001.Input.SkillInput.SkillInput3.ParameterInput.Parameterinput1.Value := 111; //TaskID
END_ACTION

ACTION Unbl111_4_exit:
//unBLOCKIEREN

Module2001.Input.SkillInput.SkillInput4.Execute := FALSE; 
Module2001.Input.SkillInput.SkillInput4.ParameterInput.Parameterinput1.Value := 000; //TaskID
END_ACTION

ACTION Unres111_5_entry:
//unreserve
Module2001.Input.SkillInput.SkillInput2.Execute := TRUE;
Module2001.Input.SkillInput.SkillInput2.ParameterInput.Parameterinput1.Value := 111; //TaskID
END_ACTION

ACTION Init_entry:
execute := FALSE;
END_ACTION

ACTION TIMER_entry:
TIMERDONE := FALSE;
END_ACTION

ACTION Unres111_5_exit:
//unreserve
Module2001.Input.SkillInput.SkillInput2.Execute := FALSE;
Module2001.Input.SkillInput.SkillInput2.ParameterInput.Parameterinput1.Value := 0; //TaskID
END_ACTION

ACTION Trans111_2_exit:
//TRANSPORTIEREN

Module2001.Input.SkillInput.SkillInput5.Execute := FALSE;
Module2001.Input.SkillInput.SkillInput5.ParameterInput.Parameterinput1.Value := 0; //X-Position
Module2001.Input.SkillInput.SkillInput5.ParameterInput.Parameterinput2.Value := 0; //Z-Position
Module2001.Input.SkillInput.SkillInput5.ParameterInput.Parameterinput3.Value := 0; //Velocity
Module2001.Input.SkillInput.SkillInput5.ParameterInput.Parameterinput4.Value := 0; //Acceleration
END_ACTION

ACTION Trans111_2_active:

END_ACTION

ACTION Res111_1_exit:
// Reservieren entry
Module2001.Input.SkillInput.SkillInput1.Execute := FALSE;
Module2001.Input.SkillInput.SkillInput1.ParameterInput.Parameterinput1.Value := 0; //TASKID
END_ACTION

END_FUNCTION_BLOCK

// ---- POUs/SkillHandle/FB_ShortTEST2.TcPOU
FUNCTION_BLOCK FB_ShortTEST2
VAR_INPUT
	execute: BOOL;
	pos2: LREAL := 2400;
END_VAR
VAR
	TIMERDONE: BOOL;
END_VAR

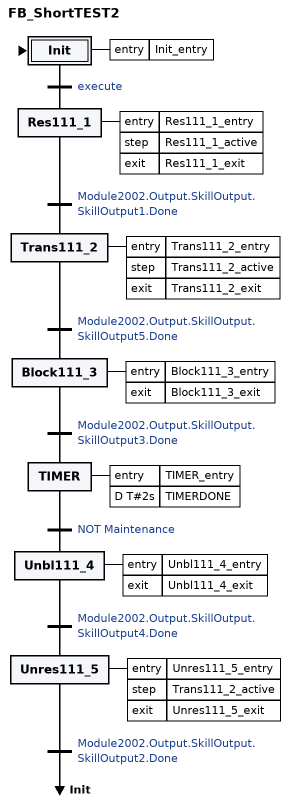
INITIAL_STEP Init:
    Init_entry(P1);  // entry action
END_STEP
TRANSITION FROM Init TO Res111_1
    := execute;
END_TRANSITION
STEP Res111_1:
    Res111_1_entry(P1);  // entry action
    Res111_1_active(N);  // step action
    Res111_1_exit(P0);  // exit action
END_STEP
TRANSITION FROM Res111_1 TO Trans111_2
    := Module2002.Output.SkillOutput.SkillOutput1.Done;
END_TRANSITION
STEP Trans111_2:
    Trans111_2_entry(P1);  // entry action
    Trans111_2_active(N);  // step action
    Trans111_2_exit(P0);  // exit action
END_STEP
TRANSITION FROM Trans111_2 TO Block111_3
    := Module2002.Output.SkillOutput.SkillOutput5.Done;
END_TRANSITION
STEP Block111_3:
    Block111_3_entry(P1);  // entry action
    Block111_3_exit(P0);  // exit action
END_STEP
TRANSITION FROM Block111_3 TO TIMER
    := Module2002.Output.SkillOutput.SkillOutput3.Done;
END_TRANSITION
STEP TIMER:
    TIMER_entry(P1);  // entry action
    TIMERDONE(D, T#2s);
END_STEP
TRANSITION FROM TIMER TO Unbl111_4
    := NOT Maintenance;
END_TRANSITION
STEP Unbl111_4:
    Unbl111_4_entry(P1);  // entry action
    Unbl111_4_exit(P0);  // exit action
END_STEP
TRANSITION FROM Unbl111_4 TO Unres111_5
    := Module2002.Output.SkillOutput.SkillOutput4.Done;
END_TRANSITION
STEP Unres111_5:
    Unres111_5_entry(P1);  // entry action
    Trans111_2_active(N);  // step action
    Unres111_5_exit(P0);  // exit action
END_STEP
TRANSITION FROM Unres111_5 TO Init
    := Module2002.Output.SkillOutput.SkillOutput2.Done;
END_TRANSITION

ACTION Res111_1_exit:
// Reservieren entry
Module2002.Input.SkillInput.SkillInput1.Execute := FALSE;
Module2002.Input.SkillInput.SkillInput1.ParameterInput.Parameterinput1.Value := 0; //TASKID
END_ACTION

ACTION Trans111_6_exit:
//TRANSPORTIEREN

Module2002.Input.SkillInput.SkillInput5.Execute := FALSE;
Module2002.Input.SkillInput.SkillInput5.ParameterInput.Parameterinput1.Value := 0; //X-Position
Module2002.Input.SkillInput.SkillInput5.ParameterInput.Parameterinput2.Value := 0; //Z-Position
Module2002.Input.SkillInput.SkillInput5.ParameterInput.Parameterinput3.Value := 0; //Velocity
Module2002.Input.SkillInput.SkillInput5.ParameterInput.Parameterinput4.Value := 0; //Acceleration
END_ACTION

ACTION Trans111_6_entry:
//TRANSPORTIEREN

Module2002.Input.SkillInput.SkillInput5.Execute := TRUE;
Module2002.Input.SkillInput.SkillInput5.ParameterInput.Parameterinput1.Value := pos2; //X-Position
Module2002.Input.SkillInput.SkillInput5.ParameterInput.Parameterinput2.Value := 80; //Z-Position
Module2002.Input.SkillInput.SkillInput5.ParameterInput.Parameterinput3.Value := 0; //Velocity
Module2002.Input.SkillInput.SkillInput5.ParameterInput.Parameterinput4.Value := 0; //Acceleration
END_ACTION

ACTION Trans111_2_entry:
//TRANSPORTIEREN

Module2002.Input.SkillInput.SkillInput5.Execute := TRUE;
Module2002.Input.SkillInput.SkillInput5.ParameterInput.Parameterinput1.Value := 1348.4; //X-Position
Module2002.Input.SkillInput.SkillInput5.ParameterInput.Parameterinput2.Value := 80; //Z-Position
Module2002.Input.SkillInput.SkillInput5.ParameterInput.Parameterinput3.Value := 0; //Velocity
Module2002.Input.SkillInput.SkillInput5.ParameterInput.Parameterinput4.Value := 0; //Acceleration
END_ACTION

ACTION Trans111_2_active:

END_ACTION

ACTION TIMER_entry:
TIMERDONE := FALSE;
END_ACTION

ACTION Unbl111_4_exit:
//unBLOCKIEREN

Module2002.Input.SkillInput.SkillInput4.Execute := FALSE; 
Module2002.Input.SkillInput.SkillInput4.ParameterInput.Parameterinput1.Value := 000; //TaskID
END_ACTION

ACTION Res111_1_active:

END_ACTION

ACTION Block111_3_exit:
//BLOCKIEREN

Module2002.Input.SkillInput.SkillInput3.Execute := FALSE;
Module2002.Input.SkillInput.SkillInput3.ParameterInput.Parameterinput1.Value := 0; //TaskID
END_ACTION

ACTION Unres111_5_entry:
//unreserve
Module2002.Input.SkillInput.SkillInput2.Execute := TRUE;
Module2002.Input.SkillInput.SkillInput2.ParameterInput.Parameterinput1.Value := 112; //TaskID
END_ACTION

ACTION Trans111_2_exit:
//TRANSPORTIEREN

Module2002.Input.SkillInput.SkillInput5.Execute := FALSE;
Module2002.Input.SkillInput.SkillInput5.ParameterInput.Parameterinput1.Value := 0; //X-Position
Module2002.Input.SkillInput.SkillInput5.ParameterInput.Parameterinput2.Value := 0; //Z-Position
Module2002.Input.SkillInput.SkillInput5.ParameterInput.Parameterinput3.Value := 0; //Velocity
Module2002.Input.SkillInput.SkillInput5.ParameterInput.Parameterinput4.Value := 0; //Acceleration
END_ACTION

ACTION Res111_1_entry:
// Reservieren entry
Module2002.Input.SkillInput.SkillInput1.Execute := TRUE;
Module2002.Input.SkillInput.SkillInput1.ParameterInput.Parameterinput1.Value := 112; //TASKID
END_ACTION

ACTION Unbl111_4_entry:
//unBLOCKIEREN

Module2002.Input.SkillInput.SkillInput4.Execute := TRUE; //FALSE weil timer
Module2002.Input.SkillInput.SkillInput4.ParameterInput.Parameterinput1.Value := 112; //TaskID
END_ACTION

ACTION Init_entry:
execute := FALSE;
END_ACTION

ACTION Block111_3_entry:
//BLOCKIEREN

Module2002.Input.SkillInput.SkillInput3.Execute := TRUE;
Module2002.Input.SkillInput.SkillInput3.ParameterInput.Parameterinput1.Value := 112; //TaskID
END_ACTION

ACTION Unres111_5_exit:
//unreserve
Module2002.Input.SkillInput.SkillInput2.Execute := FALSE;
Module2002.Input.SkillInput.SkillInput2.ParameterInput.Parameterinput1.Value := 0; //TaskID
END_ACTION

END_FUNCTION_BLOCK

// ---- POUs/SkillHandle/FB_ShortTEST3.TcPOU
FUNCTION_BLOCK FB_ShortTEST3
VAR_INPUT
	execute: BOOL;
END_VAR
VAR
	TIMERDONE: BOOL;
END_VAR

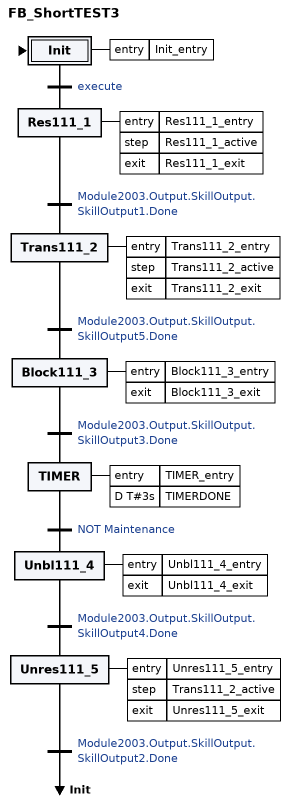
INITIAL_STEP Init:
    Init_entry(P1);  // entry action
END_STEP
TRANSITION FROM Init TO Res111_1
    := execute;
END_TRANSITION
STEP Res111_1:
    Res111_1_entry(P1);  // entry action
    Res111_1_active(N);  // step action
    Res111_1_exit(P0);  // exit action
END_STEP
TRANSITION FROM Res111_1 TO Trans111_2
    := Module2003.Output.SkillOutput.SkillOutput1.Done;
END_TRANSITION
STEP Trans111_2:
    Trans111_2_entry(P1);  // entry action
    Trans111_2_active(N);  // step action
    Trans111_2_exit(P0);  // exit action
END_STEP
TRANSITION FROM Trans111_2 TO Block111_3
    := Module2003.Output.SkillOutput.SkillOutput5.Done;
END_TRANSITION
STEP Block111_3:
    Block111_3_entry(P1);  // entry action
    Block111_3_exit(P0);  // exit action
END_STEP
TRANSITION FROM Block111_3 TO TIMER
    := Module2003.Output.SkillOutput.SkillOutput3.Done;
END_TRANSITION
STEP TIMER:
    TIMER_entry(P1);  // entry action
    TIMERDONE(D, T#3s);
END_STEP
TRANSITION FROM TIMER TO Unbl111_4
    := NOT Maintenance;
END_TRANSITION
STEP Unbl111_4:
    Unbl111_4_entry(P1);  // entry action
    Unbl111_4_exit(P0);  // exit action
END_STEP
TRANSITION FROM Unbl111_4 TO Unres111_5
    := Module2003.Output.SkillOutput.SkillOutput4.Done;
END_TRANSITION
STEP Unres111_5:
    Unres111_5_entry(P1);  // entry action
    Trans111_2_active(N);  // step action
    Unres111_5_exit(P0);  // exit action
END_STEP
TRANSITION FROM Unres111_5 TO Init
    := Module2003.Output.SkillOutput.SkillOutput2.Done;
END_TRANSITION

ACTION Unres111_5_exit:
//unreserve
Module2003.Input.SkillInput.SkillInput2.Execute := FALSE;
Module2003.Input.SkillInput.SkillInput2.ParameterInput.Parameterinput1.Value := 0; //TaskID
END_ACTION

ACTION Block111_3_entry:
//BLOCKIEREN

Module2003.Input.SkillInput.SkillInput3.Execute := TRUE;
Module2003.Input.SkillInput.SkillInput3.ParameterInput.Parameterinput1.Value := 113; //TaskID
END_ACTION

ACTION Res111_1_active:

END_ACTION

ACTION Trans111_2_active:

END_ACTION

ACTION Trans111_2_entry:
//TRANSPORTIEREN

Module2003.Input.SkillInput.SkillInput5.Execute := TRUE;
Module2003.Input.SkillInput.SkillInput5.ParameterInput.Parameterinput1.Value := 169.4; //X-Position
Module2003.Input.SkillInput.SkillInput5.ParameterInput.Parameterinput2.Value := 90; //Z-Position
Module2003.Input.SkillInput.SkillInput5.ParameterInput.Parameterinput3.Value := 400; //Velocity
Module2003.Input.SkillInput.SkillInput5.ParameterInput.Parameterinput4.Value := 100; //Acceleration
END_ACTION

ACTION Unres111_5_entry:
//unreserve
Module2003.Input.SkillInput.SkillInput2.Execute := TRUE;
Module2003.Input.SkillInput.SkillInput2.ParameterInput.Parameterinput1.Value := 113; //TaskID
END_ACTION

ACTION Trans111_6_entry:
//TRANSPORTIEREN

Module2003.Input.SkillInput.SkillInput5.Execute := TRUE;
Module2003.Input.SkillInput.SkillInput5.ParameterInput.Parameterinput1.Value := 20; //X-Position
Module2003.Input.SkillInput.SkillInput5.ParameterInput.Parameterinput2.Value := 80; //Z-Position
Module2003.Input.SkillInput.SkillInput5.ParameterInput.Parameterinput3.Value := 0; //Velocity
Module2003.Input.SkillInput.SkillInput5.ParameterInput.Parameterinput4.Value := 0; //Acceleration
END_ACTION

ACTION Trans111_2_exit:
//TRANSPORTIEREN

Module2003.Input.SkillInput.SkillInput5.Execute := FALSE;
Module2003.Input.SkillInput.SkillInput5.ParameterInput.Parameterinput1.Value := 0; //X-Position
Module2003.Input.SkillInput.SkillInput5.ParameterInput.Parameterinput2.Value := 0; //Z-Position
Module2003.Input.SkillInput.SkillInput5.ParameterInput.Parameterinput3.Value := 0; //Velocity
Module2003.Input.SkillInput.SkillInput5.ParameterInput.Parameterinput4.Value := 0; //Acceleration
END_ACTION

ACTION Init_entry:
execute := FALSE;
END_ACTION

ACTION Res111_1_exit:
// Reservieren entry
Module2003.Input.SkillInput.SkillInput1.Execute := FALSE;
Module2003.Input.SkillInput.SkillInput1.ParameterInput.Parameterinput1.Value := 0; //TASKID
END_ACTION

ACTION TIMER_entry:
TIMERDONE := FALSE;
END_ACTION

ACTION Unbl111_4_entry:
//unBLOCKIEREN

Module2003.Input.SkillInput.SkillInput4.Execute := TRUE; //FALSE weil timer
Module2003.Input.SkillInput.SkillInput4.ParameterInput.Parameterinput1.Value := 112; //TaskID
END_ACTION

ACTION Unbl111_4_exit:
//unBLOCKIEREN

Module2003.Input.SkillInput.SkillInput4.Execute := FALSE; 
Module2003.Input.SkillInput.SkillInput4.ParameterInput.Parameterinput1.Value := 000; //TaskID
END_ACTION

ACTION Trans111_6_exit:
//TRANSPORTIEREN

Module2003.Input.SkillInput.SkillInput5.Execute := FALSE;
Module2003.Input.SkillInput.SkillInput5.ParameterInput.Parameterinput1.Value := 0; //X-Position
Module2003.Input.SkillInput.SkillInput5.ParameterInput.Parameterinput2.Value := 0; //Z-Position
Module2003.Input.SkillInput.SkillInput5.ParameterInput.Parameterinput3.Value := 0; //Velocity
Module2003.Input.SkillInput.SkillInput5.ParameterInput.Parameterinput4.Value := 0; //Acceleration
END_ACTION

ACTION Res111_1_entry:
// Reservieren entry
Module2003.Input.SkillInput.SkillInput1.Execute := TRUE;
Module2003.Input.SkillInput.SkillInput1.ParameterInput.Parameterinput1.Value := 113; //TASKID
END_ACTION

ACTION Block111_3_exit:
//BLOCKIEREN

Module2003.Input.SkillInput.SkillInput3.Execute := FALSE;
Module2003.Input.SkillInput.SkillInput3.ParameterInput.Parameterinput1.Value := 0; //TaskID
END_ACTION

END_FUNCTION_BLOCK

// ---- POUs/SkillHandle/FB_2001_cocktail.TcPOU
FUNCTION_BLOCK FB_2001_cocktail
VAR_INPUT
	execute: BOOL;
END_VAR
VAR
	TIMERDONE: BOOL;
END_VAR

